LIN {X 0,Y 203.578,Z 1003.73,A -85,B 0,C 180,E1 8716.654,E2 8716.654} C_VEL
LIN {X 0,Y 203.632,Z 1006.005,A -85,B 0,C 180,E1 8711.685,E2 8711.685} C_VEL
LIN {X 0,Y 204.624,Z 1006.572,A -85,B 0,C 180,E1 8706.685,E2 8706.685} C_VEL
LIN {X 0,Y 206.666,Z 1005.305,A -85,B 0,C 180,E1 8701.698,E2 8701.698} C_VEL
LIN {X 0,Y 209.886,Z 1002.177,A -85,B 0,C 180,E1 8696.782,E2 8696.782} C_VEL
LIN {X 0,Y 214.071,Z 997.405,A -85,B 0,C 180,E1 8692.277,E2 8692.277} C_VEL
LIN {X 0,Y 219.005,Z 991.1,A -85,B 0,C 180,E1 8688.199,E2 8688.199} C_VEL
LIN {X 0,Y 224.873,Z 982.735,A -85,B 0,C 180,E1 8684.287,E2 8684.287} C_VEL
LIN {X 0,Y 231.227,Z 972.677,A -85,B 0,C 180,E1 8680.765,E2 8680.765} C_VEL
LIN {X 0,Y 237.626,Z 961.261,A -85,B 0,C 180,E1 8677.717,E2 8677.717} C_VEL
LIN {X 0,Y 243.815,Z 948.504,A -85,B 0,C 180,E1 8675.103,E2 8675.103} C_VEL
LIN {X 0,Y 249.813,Z 934.055,A -85,B 0,C 180,E1 8672.807,E2 8672.807} C_VEL
LIN {X 0,Y 254.885,Z 919.39,A -85,B 0,C 180,E1 8671.005,E2 8671.005} C_VEL
LIN {X 0,Y 259.318,Z 903.23,A -85,B 0,C 180,E1 8669.492,E2 8669.492} C_VEL
LIN {X 0,Y 262.776,Z 886.237,A -85,B 0,C 180,E1 8668.313,E2 8668.313} C_VEL
LIN {X 0,Y 265.149,Z 868.666,A -85,B 0,C 180,E1 8667.459,E2 8667.459} C_VEL
LIN {X 0,Y 267.85,Z 833.08,A -85,B 0,C 180,E1 8666.452,E2 8666.452} C_VEL
LIN {X 0,Y 269.767,Z 808.526,A -85,B 0,C 180,E1 8665.844,E2 8665.844} C_VEL
LIN {X 0,Y 269.834,Z 800.953,A -85,B 0,C 180,E1 8665.478,E2 8665.478} C_VEL
LIN {X 0,Y 268.193,Z 781.182,A -85,B 0,C 180,E1 8663.856,E2 8663.856} C_VEL
LIN {X 0,Y 268.351,Z 774.67,A -85,B 0,C 180,E1 8663.562,E2 8663.562} C_VEL
LIN {X 0,Y 268.8,Z 767.997,A -85,B 0,C 180,E1 8663.367,E2 8663.367} C_VEL
LIN {X 0,Y 263.509,Z 757.018,A -85,B 0,C 180,E1 8660.606,E2 8660.606} C_VEL
LIN {X 0,Y 258.076,Z 747.072,A -85,B 0,C 180,E1 8657.415,E2 8657.415} C_VEL
LIN {X 0,Y 253.684,Z 739.87,A -85,B 0,C 180,E1 8654.378,E2 8654.378} C_VEL
LIN {X 0,Y 250.818,Z 735.384,A -85,B 0,C 180,E1 8652.081,E2 8652.081} C_VEL
LIN {X 0,Y 246.984,Z 729.389,A -85,B 0,C 180,E1 8648.263,E2 8648.263} C_VEL
LIN {X 0,Y 243.777,Z 724.701,A -85,B 0,C 180,E1 8643.763,E2 8643.763} C_VEL
LIN {X 0,Y 241.598,Z 721.587,A -85,B 0,C 180,E1 8637.391,E2 8637.391} C_VEL
LIN {X 0,Y 241.91,Z 721.898,A -85,B 0,C 180,E1 8631.922,E2 8631.922} C_VEL
LIN {X 0,Y 245.181,Z 726.188,A -85,B 0,C 180,E1 8624.992,E2 8624.992} C_VEL
LIN {X 0,Y 249.877,Z 733.151,A -85,B 0,C 180,E1 8619.75,E2 8619.75} C_VEL
LIN {X 0,Y 254.492,Z 740.242,A -85,B 0,C 180,E1 8616.007,E2 8616.007} C_VEL
LIN {X 0,Y 259.061,Z 747.772,A -85,B 0,C 180,E1 8612.97,E2 8612.97} C_VEL
LIN {X 0,Y 263.465,Z 755.393,A -85,B 0,C 180,E1 8610.439,E2 8610.439} C_VEL
LIN {X 0,Y 268.804,Z 765.811,A -85,B 0,C 180,E1 8607.677,E2 8607.677} C_VEL
LIN {X 0,Y 269.518,Z 767.79,A -85,B 0,C 180,E1 8607.302,E2 8607.302} C_VEL
LIN {X 0,Y 259.299,Z 896.401,A -85,B 0,C 180,E1 8604.125,E2 8604.125} C_VEL
LIN {X 0,Y 256.355,Z 915.058,A -85,B 0,C 180,E1 8603.402,E2 8603.402} C_VEL
LIN {X 0,Y 252.244,Z 932.623,A -85,B 0,C 180,E1 8602.444,E2 8602.444} C_VEL
LIN {X 0,Y 246.71,Z 950.675,A -85,B 0,C 180,E1 8601.089,E2 8601.089} C_VEL
LIN {X 0,Y 240.772,Z 966.702,A -85,B 0,C 180,E1 8599.459,E2 8599.459} C_VEL
LIN {X 0,Y 234.223,Z 981.979,A -85,B 0,C 180,E1 8597.423,E2 8597.423} C_VEL
LIN {X 0,Y 227.206,Z 996.499,A -85,B 0,C 180,E1 8594.917,E2 8594.917} C_VEL
LIN {X 0,Y 220.048,Z 1010.012,A -85,B 0,C 180,E1 8591.908,E2 8591.908} C_VEL
LIN {X 0,Y 212.964,Z 1022.543,A -85,B 0,C 180,E1 8588.296,E2 8588.296} C_VEL
LIN {X 0,Y 206.391,Z 1033.8,A -85,B 0,C 180,E1 8584.065,E2 8584.065} C_VEL
LIN {X 0,Y 201.054,Z 1043.16,A -85,B 0,C 180,E1 8579.493,E2 8579.493} C_VEL
LIN {X 0,Y 196.839,Z 1051.262,A -85,B 0,C 180,E1 8574.295,E2 8574.295} C_VEL
LIN {X 0,Y 194.203,Z 1057.772,A -85,B 0,C 180,E1 8568.614,E2 8568.614} C_VEL
LIN {X 0,Y 193.286,Z 1062.33,A -85,B 0,C 180,E1 8562.851,E2 8562.851} C_VEL
LIN {X 0,Y 193.748,Z 1064.894,A -85,B 0,C 180,E1 8557.412,E2 8557.412} C_VEL
LIN {X 0,Y 194.69,Z 1065.679,A -85,B 0,C 180,E1 8552.648,E2 8552.648} C_VEL
LIN {X 0,Y 194.99,Z 1065.259,A -85,B 0,C 180,E1 8549.118,E2 8549.118} C_VEL
LIN {X 0,Y 194.449,Z 1063.524,A -85,B 0,C 180,E1 8544.984,E2 8544.984} C_VEL
LIN {X 0,Y 193.509,Z 1061.492,A -85,B 0,C 180,E1 8539.279,E2 8539.279} C_VEL
LIN {X 0,Y 193.709,Z 1057.837,A -85,B 0,C 180,E1 8534.122,E2 8534.122} C_VEL
LIN {X 0,Y 195.37,Z 1051.854,A -85,B 0,C 180,E1 8528.692,E2 8528.692} C_VEL
LIN {X 0,Y 198.492,Z 1044.215,A -85,B 0,C 180,E1 8523.686,E2 8523.686} C_VEL
LIN {X 0,Y 203.06,Z 1034.434,A -85,B 0,C 180,E1 8518.867,E2 8518.867} C_VEL
LIN {X 0,Y 208.337,Z 1023.844,A -85,B 0,C 180,E1 8514.836,E2 8514.836} C_VEL
LIN {X 0,Y 214.759,Z 1011.017,A -85,B 0,C 180,E1 8511.058,E2 8511.058} C_VEL
LIN {X 0,Y 221.183,Z 997.712,A -85,B 0,C 180,E1 8508.006,E2 8508.006} C_VEL
LIN {X 0,Y 228.022,Z 982.335,A -85,B 0,C 180,E1 8505.264,E2 8505.264} C_VEL
LIN {X 0,Y 234.291,Z 966.649,A -85,B 0,C 180,E1 8503.133,E2 8503.133} C_VEL
LIN {X 0,Y 240.05,Z 949.931,A -85,B 0,C 180,E1 8501.431,E2 8501.431} C_VEL
LIN {X 0,Y 244.754,Z 933.123,A -85,B 0,C 180,E1 8500.21,E2 8500.21} C_VEL
LIN {X 0,Y 248.664,Z 914.35,A -85,B 0,C 180,E1 8499.236,E2 8499.236} C_VEL
LIN {X 0,Y 268.436,Z 803.055,A -85,B 0,C 180,E1 8494.981,E2 8494.981} C_VEL
LIN {X 0,Y 273.515,Z 775.803,A -85,B 0,C 180,E1 8493.883,E2 8493.883} C_VEL
LIN {X 0,Y 274.688,Z 769.516,A -85,B 0,C 180,E1 8493.533,E2 8493.533} C_VEL
LIN {X 0,Y 276.759,Z 763.473,A -85,B 0,C 180,E1 8492.948,E2 8492.948} C_VEL
LIN {X 0,Y 277.255,Z 762.029,A -85,B 0,C 180,E1 8492.448,E2 8492.448} C_VEL
LIN {X 0,Y 276.155,Z 764.633,A -85,B 0,C 180,E1 8490.216,E2 8490.216} C_VEL
LIN {X 0,Y 276.372,Z 769.354,A -85,B 0,C 180,E1 8488.054,E2 8488.054} C_VEL
LIN {X 0,Y 276.354,Z 770.749,A -85,B 0,C 180,E1 8487.719,E2 8487.719} C_VEL
LIN {X 0,Y 276.091,Z 773.303,A -85,B 0,C 180,E1 8487.445,E2 8487.445} C_VEL
LIN {X 0,Y 260.146,Z 869.807,A -85,B 0,C 180,E1 8483.989,E2 8483.989} C_VEL
LIN {X 0,Y 255.611,Z 901.484,A -85,B 0,C 180,E1 8482.427,E2 8482.427} C_VEL
LIN {X 0,Y 252.75,Z 916.861,A -85,B 0,C 180,E1 8481.342,E2 8481.342} C_VEL
LIN {X 0,Y 248.618,Z 932.379,A -85,B 0,C 180,E1 8479.866,E2 8479.866} C_VEL
LIN {X 0,Y 243.925,Z 946.223,A -85,B 0,C 180,E1 8478.151,E2 8478.151} C_VEL
LIN {X 0,Y 238.087,Z 960.158,A -85,B 0,C 180,E1 8475.907,E2 8475.907} C_VEL
LIN {X 0,Y 232.173,Z 971.846,A -85,B 0,C 180,E1 8473.447,E2 8473.447} C_VEL
LIN {X 0,Y 226.238,Z 982.029,A -85,B 0,C 180,E1 8470.697,E2 8470.697} C_VEL
LIN {X 0,Y 219.74,Z 991.542,A -85,B 0,C 180,E1 8467.273,E2 8467.273} C_VEL
LIN {X 0,Y 214.041,Z 998.695,A -85,B 0,C 180,E1 8463.749,E2 8463.749} C_VEL
LIN {X 0,Y 208.667,Z 1004.435,A -85,B 0,C 180,E1 8459.725,E2 8459.725} C_VEL
LIN {X 0,Y 204.19,Z 1008.247,A -85,B 0,C 180,E1 8455.506,E2 8455.506} C_VEL
LIN {X 0,Y 200.448,Z 1010.368,A -85,B 0,C 180,E1 8450.815,E2 8450.815} C_VEL
LIN {X 0,Y 197.801,Z 1010.466,A -85,B 0,C 180,E1 8446.061,E2 8446.061} C_VEL
LIN {X 0,Y 196.221,Z 1008.801,A -85,B 0,C 180,E1 8441.404,E2 8441.404} C_VEL
LIN {X 0,Y 195.451,Z 1005.065,A -85,B 0,C 180,E1 8436.482,E2 8436.482} C_VEL
LIN {X 0,Y 195.491,Z 999.785,A -85,B 0,C 180,E1 8431.93,E2 8431.93} C_VEL
LIN {X 0,Y 196.255,Z 992.329,A -85,B 0,C 180,E1 8427.313,E2 8427.313} C_VEL
LIN {X 0,Y 197.544,Z 983.866,A -85,B 0,C 180,E1 8423.326,E2 8423.326} C_VEL
LIN {X 0,Y 199.467,Z 973.093,A -85,B 0,C 180,E1 8419.333,E2 8419.333} C_VEL
LIN {X 0,Y 201.823,Z 960.491,A -85,B 0,C 180,E1 8415.69,E2 8415.69} C_VEL
LIN {X 0,Y 204.168,Z 947.545,A -85,B 0,C 180,E1 8412.727,E2 8412.727} C_VEL
LIN {X 0,Y 206.602,Z 932.888,A -85,B 0,C 180,E1 8410.066,E2 8410.066} C_VEL
LIN {X 0,Y 208.893,Z 916.417,A -85,B 0,C 180,E1 8407.784,E2 8407.784} C_VEL
LIN {X 0,Y 210.657,Z 900.18,A -85,B 0,C 180,E1 8406.102,E2 8406.102} C_VEL
LIN {X 0,Y 211.969,Z 882.792,A -85,B 0,C 180,E1 8404.823,E2 8404.823} C_VEL
LIN {X 0,Y 214.763,Z 828.021,A -85,B 0,C 180,E1 8402.341,E2 8402.341} C_VEL
LIN {X 0,Y 217.097,Z 797.981,A -85,B 0,C 180,E1 8400.978,E2 8400.978} C_VEL
LIN {X 0,Y 218.251,Z 792.429,A -85,B 0,C 180,E1 8400.462,E2 8400.462} C_VEL
LIN {X 0,Y 220.656,Z 789.756,A -85,B 0,C 180,E1 8399.866,E2 8399.866} C_VEL
LIN {X 0,Y 223.732,Z 783.211,A -85,B 0,C 180,E1 8399.37,E2 8399.37} C_VEL
LIN {X 0,Y 228.317,Z 768.728,A -85,B 0,C 180,E1 8398.869,E2 8398.869} C_VEL
LIN {X 0,Y 232.213,Z 755.083,A -85,B 0,C 180,E1 8398.519,E2 8398.519} C_VEL
LIN {X 0,Y 236.759,Z 749.133,A -85,B 0,C 180,E1 8397.714,E2 8397.714} C_VEL
LIN {X 0,Y 237.715,Z 747.772,A -85,B 0,C 180,E1 8397.554,E2 8397.554} C_VEL
LIN {X 0,Y 238.404,Z 755.137,A -85,B 0,C 180,E1 8397.101,E2 8397.101} C_VEL
LIN {X 0,Y 232.035,Z 861.838,A -85,B 0,C 180,E1 8394.081,E2 8394.081} C_VEL
LIN {X 0,Y 230.476,Z 879.542,A -85,B 0,C 180,E1 8393.202,E2 8393.202} C_VEL
LIN {X 0,Y 228.187,Z 895.686,A -85,B 0,C 180,E1 8392.003,E2 8392.003} C_VEL
LIN {X 0,Y 224.933,Z 912.565,A -85,B 0,C 180,E1 8390.288,E2 8390.288} C_VEL
LIN {X 0,Y 221.154,Z 928.279,A -85,B 0,C 180,E1 8388.178,E2 8388.178} C_VEL
LIN {X 0,Y 217.076,Z 942.488,A -85,B 0,C 180,E1 8385.705,E2 8385.705} C_VEL
LIN {X 0,Y 212.77,Z 955.748,A -85,B 0,C 180,E1 8382.761,E2 8382.761} C_VEL
LIN {X 0,Y 208.516,Z 967.742,A -85,B 0,C 180,E1 8379.384,E2 8379.384} C_VEL
LIN {X 0,Y 204.574,Z 978.262,A -85,B 0,C 180,E1 8375.61,E2 8375.61} C_VEL
LIN {X 0,Y 201.023,Z 987.567,A -85,B 0,C 180,E1 8371.263,E2 8371.263} C_VEL
LIN {X 0,Y 198.271,Z 995.222,A -85,B 0,C 180,E1 8366.531,E2 8366.531} C_VEL
LIN {X 0,Y 196.546,Z 1000.808,A -85,B 0,C 180,E1 8361.812,E2 8361.812} C_VEL
LIN {X 0,Y 195.657,Z 1004.859,A -85,B 0,C 180,E1 8356.706,E2 8356.706} C_VEL
LIN {X 0,Y 195.725,Z 1007.171,A -85,B 0,C 180,E1 8351.536,E2 8351.536} C_VEL
LIN {X 0,Y 196.795,Z 1007.783,A -85,B 0,C 180,E1 8346.337,E2 8346.337} C_VEL
LIN {X 0,Y 198.981,Z 1006.591,A -85,B 0,C 180,E1 8341.159,E2 8341.159} C_VEL
LIN {X 0,Y 202.406,Z 1003.52,A -85,B 0,C 180,E1 8336.069,E2 8336.069} C_VEL
LIN {X 0,Y 206.835,Z 998.812,A -85,B 0,C 180,E1 8331.421,E2 8331.421} C_VEL
LIN {X 0,Y 212.033,Z 992.609,A -85,B 0,C 180,E1 8327.232,E2 8327.232} C_VEL
LIN {X 0,Y 218.188,Z 984.347,A -85,B 0,C 180,E1 8323.229,E2 8323.229} C_VEL
LIN {X 0,Y 224.746,Z 974.521,A -85,B 0,C 180,E1 8319.679,E2 8319.679} C_VEL
LIN {X 0,Y 231.49,Z 963.14,A -85,B 0,C 180,E1 8316.547,E2 8316.547} C_VEL
LIN {X 0,Y 238.009,Z 950.434,A -85,B 0,C 180,E1 8313.872,E2 8313.872} C_VEL
LIN {X 0,Y 244.144,Z 936.403,A -85,B 0,C 180,E1 8311.589,E2 8311.589} C_VEL
LIN {X 0,Y 249.711,Z 921.122,A -85,B 0,C 180,E1 8309.672,E2 8309.672} C_VEL
LIN {X 0,Y 254.364,Z 905.152,A -85,B 0,C 180,E1 8308.145,E2 8308.145} C_VEL
LIN {X 0,Y 258.014,Z 888.279,A -85,B 0,C 180,E1 8306.949,E2 8306.949} C_VEL
LIN {X 0,Y 260.608,Z 870.365,A -85,B 0,C 180,E1 8306.056,E2 8306.056} C_VEL
LIN {X 0,Y 262.922,Z 841.507,A -85,B 0,C 180,E1 8305.196,E2 8305.196} C_VEL
LIN {X 0,Y 268.351,Z 774.67,A -85,B 0,C 180,E1 8303.562,E2 8303.562} C_VEL
LIN {X 0,Y 268.12,Z 771.832,A -85,B 0,C 180,E1 8303.321,E2 8303.321} C_VEL
LIN {X 0,Y 266.748,Z 768.797,A -85,B 0,C 180,E1 8302.625,E2 8302.625} C_VEL
LIN {X 0,Y 263.914,Z 766.213,A -85,B 0,C 180,E1 8301.332,E2 8301.332} C_VEL
LIN {X 0,Y 260.671,Z 763.319,A -85,B 0,C 180,E1 8299.747,E2 8299.747} C_VEL
LIN {X 0,Y 260.14,Z 762.462,A -85,B 0,C 180,E1 8299.45,E2 8299.45} C_VEL
LIN {X 0,Y 255.618,Z 753.768,A -85,B 0,C 180,E1 8296.592,E2 8296.592} C_VEL
LIN {X 0,Y 251.564,Z 746.869,A -85,B 0,C 180,E1 8293.621,E2 8293.621} C_VEL
LIN {X 0,Y 248.889,Z 742.531,A -85,B 0,C 180,E1 8291.353,E2 8291.353} C_VEL
LIN {X 0,Y 245.454,Z 736.952,A -85,B 0,C 180,E1 8287.726,E2 8287.726} C_VEL
LIN {X 0,Y 242.497,Z 732.417,A -85,B 0,C 180,E1 8283.31,E2 8283.31} C_VEL
LIN {X 0,Y 240.565,Z 729.488,A -85,B 0,C 180,E1 8277.142,E2 8277.142} C_VEL
LIN {X 0,Y 240.896,Z 729.875,A -85,B 0,C 180,E1 8271.888,E2 8271.888} C_VEL
LIN {X 0,Y 243.919,Z 734.075,A -85,B 0,C 180,E1 8265.277,E2 8265.277} C_VEL
LIN {X 0,Y 248.264,Z 740.711,A -85,B 0,C 180,E1 8260.227,E2 8260.227} C_VEL
LIN {X 0,Y 252.592,Z 747.658,A -85,B 0,C 180,E1 8256.559,E2 8256.559} C_VEL
LIN {X 0,Y 256.823,Z 754.954,A -85,B 0,C 180,E1 8253.59,E2 8253.59} C_VEL
LIN {X 0,Y 261.285,Z 762.982,A -85,B 0,C 180,E1 8250.923,E2 8250.923} C_VEL
LIN {X 0,Y 265.322,Z 771.367,A -85,B 0,C 180,E1 8248.717,E2 8248.717} C_VEL
LIN {X 0,Y 255.038,Z 895.526,A -85,B 0,C 180,E1 8245.649,E2 8245.649} C_VEL
LIN {X 0,Y 251.997,Z 914.175,A -85,B 0,C 180,E1 8244.931,E2 8244.931} C_VEL
LIN {X 0,Y 247.449,Z 932.835,A -85,B 0,C 180,E1 8243.913,E2 8243.913} C_VEL
LIN {X 0,Y 242.101,Z 949.634,A -85,B 0,C 180,E1 8242.655,E2 8242.655} C_VEL
LIN {X 0,Y 235.949,Z 965.673,A -85,B 0,C 180,E1 8241.04,E2 8241.04} C_VEL
LIN {X 0,Y 229.144,Z 980.95,A -85,B 0,C 180,E1 8239.014,E2 8239.014} C_VEL
LIN {X 0,Y 221.852,Z 995.407,A -85,B 0,C 180,E1 8236.519,E2 8236.519} C_VEL
LIN {X 0,Y 214.049,Z 1009.428,A -85,B 0,C 180,E1 8233.366,E2 8233.366} C_VEL
LIN {X 0,Y 206.548,Z 1021.914,A -85,B 0,C 180,E1 8229.675,E2 8229.675} C_VEL
LIN {X 0,Y 199.783,Z 1032.778,A -85,B 0,C 180,E1 8225.488,E2 8225.488} C_VEL
LIN {X 0,Y 193.93,Z 1042.278,A -85,B 0,C 180,E1 8220.691,E2 8220.691} C_VEL
LIN {X 0,Y 189.366,Z 1050.289,A -85,B 0,C 180,E1 8215.32,E2 8215.32} C_VEL
LIN {X 0,Y 186.435,Z 1056.73,A -85,B 0,C 180,E1 8209.42,E2 8209.42} C_VEL
LIN {X 0,Y 185.341,Z 1061.223,A -85,B 0,C 180,E1 8203.412,E2 8203.412} C_VEL
LIN {X 0,Y 185.749,Z 1063.725,A -85,B 0,C 180,E1 8197.733,E2 8197.733} C_VEL
LIN {X 0,Y 186.751,Z 1064.458,A -85,B 0,C 180,E1 8192.761,E2 8192.761} C_VEL
LIN {X 0,Y 187.081,Z 1064.008,A -85,B 0,C 180,E1 8189.08,E2 8189.08} C_VEL
LIN {X 0,Y 186.484,Z 1062.177,A -85,B 0,C 180,E1 8184.77,E2 8184.77} C_VEL
LIN {X 0,Y 185.543,Z 1060.5,A -85,B 0,C 180,E1 8179.128,E2 8179.128} C_VEL
LIN {X 0,Y 185.831,Z 1056.902,A -85,B 0,C 180,E1 8173.43,E2 8173.43} C_VEL
LIN {X 0,Y 187.608,Z 1051.546,A -85,B 0,C 180,E1 8168.022,E2 8168.022} C_VEL
LIN {X 0,Y 191.174,Z 1043.948,A -85,B 0,C 180,E1 8162.596,E2 8162.596} C_VEL
LIN {X 0,Y 195.809,Z 1035.264,A -85,B 0,C 180,E1 8157.922,E2 8157.922} C_VEL
LIN {X 0,Y 201.824,Z 1024.535,A -85,B 0,C 180,E1 8153.522,E2 8153.522} C_VEL
LIN {X 0,Y 208.687,Z 1012.412,A -85,B 0,C 180,E1 8149.698,E2 8149.698} C_VEL
LIN {X 0,Y 216.326,Z 998.234,A -85,B 0,C 180,E1 8146.291,E2 8146.291} C_VEL
LIN {X 0,Y 223.322,Z 984.22,A -85,B 0,C 180,E1 8143.691,E2 8143.691} C_VEL
LIN {X 0,Y 230.618,Z 967.927,A -85,B 0,C 180,E1 8141.404,E2 8141.404} C_VEL
LIN {X 0,Y 236.718,Z 952.148,A -85,B 0,C 180,E1 8139.758,E2 8139.758} C_VEL
LIN {X 0,Y 242.101,Z 935.373,A -85,B 0,C 180,E1 8138.498,E2 8138.498} C_VEL
LIN {X 0,Y 246.595,Z 916.793,A -85,B 0,C 180,E1 8137.514,E2 8137.514} C_VEL
LIN {X 0,Y 253.262,Z 880.318,A -85,B 0,C 180,E1 8136.065,E2 8136.065} C_VEL
LIN {X 0,Y 270.986,Z 787.896,A -85,B 0,C 180,E1 8132.689,E2 8132.689} C_VEL
LIN {X 0,Y 274.114,Z 772.366,A -85,B 0,C 180,E1 8131.977,E2 8131.977} C_VEL
LIN {X 0,Y 274.515,Z 770.48,A -85,B 0,C 180,E1 8131.791,E2 8131.791} C_VEL
LIN {X 0,Y 274.43,Z 774.056,A -85,B 0,C 180,E1 8129.703,E2 8129.703} C_VEL
LIN {X 0,Y 274.437,Z 775.934,A -85,B 0,C 180,E1 8129.019,E2 8129.019} C_VEL
LIN {X 0,Y 257.896,Z 870.774,A -85,B 0,C 180,E1 8125.674,E2 8125.674} C_VEL
LIN {X 0,Y 252.941,Z 902.761,A -85,B 0,C 180,E1 8124.102,E2 8124.102} C_VEL
LIN {X 0,Y 249.734,Z 918.743,A -85,B 0,C 180,E1 8122.977,E2 8122.977} C_VEL
LIN {X 0,Y 245.337,Z 934.072,A -85,B 0,C 180,E1 8121.517,E2 8121.517} C_VEL
LIN {X 0,Y 240.351,Z 947.81,A -85,B 0,C 180,E1 8119.818,E2 8119.818} C_VEL
LIN {X 0,Y 233.955,Z 962.022,A -85,B 0,C 180,E1 8117.522,E2 8117.522} C_VEL
LIN {X 0,Y 227.02,Z 974.708,A -85,B 0,C 180,E1 8114.8,E2 8114.8} C_VEL
LIN {X 0,Y 220.693,Z 984.536,A -85,B 0,C 180,E1 8112.028,E2 8112.028} C_VEL
LIN {X 0,Y 213.872,Z 993.716,A -85,B 0,C 180,E1 8108.603,E2 8108.603} C_VEL
LIN {X 0,Y 207.285,Z 1001.173,A -85,B 0,C 180,E1 8104.703,E2 8104.703} C_VEL
LIN {X 0,Y 201.577,Z 1006.585,A -85,B 0,C 180,E1 8100.568,E2 8100.568} C_VEL
LIN {X 0,Y 196.529,Z 1010.278,A -85,B 0,C 180,E1 8095.915,E2 8095.915} C_VEL
LIN {X 0,Y 192.812,Z 1011.909,A -85,B 0,C 180,E1 8091.35,E2 8091.35} C_VEL
LIN {X 0,Y 189.944,Z 1011.756,A -85,B 0,C 180,E1 8086.297,E2 8086.297} C_VEL
LIN {X 0,Y 188.266,Z 1009.727,A -85,B 0,C 180,E1 8081.418,E2 8081.418} C_VEL
LIN {X 0,Y 187.491,Z 1005.848,A -85,B 0,C 180,E1 8076.423,E2 8076.423} C_VEL
LIN {X 0,Y 187.545,Z 1000.16,A -85,B 0,C 180,E1 8071.604,E2 8071.604} C_VEL
LIN {X 0,Y 188.331,Z 992.822,A -85,B 0,C 180,E1 8067.018,E2 8067.018} C_VEL
LIN {X 0,Y 189.761,Z 983.773,A -85,B 0,C 180,E1 8062.703,E2 8062.703} C_VEL
LIN {X 0,Y 191.624,Z 973.621,A -85,B 0,C 180,E1 8058.894,E2 8058.894} C_VEL
LIN {X 0,Y 194.087,Z 960.838,A -85,B 0,C 180,E1 8055.107,E2 8055.107} C_VEL
LIN {X 0,Y 196.671,Z 946.905,A -85,B 0,C 180,E1 8051.884,E2 8051.884} C_VEL
LIN {X 0,Y 199.111,Z 932.453,A -85,B 0,C 180,E1 8049.252,E2 8049.252} C_VEL
LIN {X 0,Y 201.448,Z 916.135,A -85,B 0,C 180,E1 8046.955,E2 8046.955} C_VEL
LIN {X 0,Y 203.406,Z 898.223,A -85,B 0,C 180,E1 8045.109,E2 8045.109} C_VEL
LIN {X 0,Y 204.686,Z 880.46,A -85,B 0,C 180,E1 8043.857,E2 8043.857} C_VEL
LIN {X 0,Y 206.821,Z 840.303,A -85,B 0,C 180,E1 8041.878,E2 8041.878} C_VEL
LIN {X 0,Y 207.906,Z 834.54,A -85,B 0,C 180,E1 8041.317,E2 8041.317} C_VEL
LIN {X 0,Y 210.557,Z 831.512,A -85,B 0,C 180,E1 8040.604,E2 8040.604} C_VEL
LIN {X 0,Y 213.729,Z 824.641,A -85,B 0,C 180,E1 8040.064,E2 8040.064} C_VEL
LIN {X 0,Y 218.392,Z 809.936,A -85,B 0,C 180,E1 8039.521,E2 8039.521} C_VEL
LIN {X 0,Y 221.875,Z 797.999,A -85,B 0,C 180,E1 8039.176,E2 8039.176} C_VEL
LIN {X 0,Y 225.197,Z 793.883,A -85,B 0,C 180,E1 8038.531,E2 8038.531} C_VEL
LIN {X 0,Y 228.812,Z 786.166,A -85,B 0,C 180,E1 8037.996,E2 8037.996} C_VEL
LIN {X 0,Y 230.951,Z 780.277,A -85,B 0,C 180,E1 8037.746,E2 8037.746} C_VEL
LIN {X 0,Y 225.842,Z 863.105,A -85,B 0,C 180,E1 8035.328,E2 8035.328} C_VEL
LIN {X 0,Y 224.174,Z 880.79,A -85,B 0,C 180,E1 8034.42,E2 8034.42} C_VEL
LIN {X 0,Y 221.612,Z 897.765,A -85,B 0,C 180,E1 8033.112,E2 8033.112} C_VEL
LIN {X 0,Y 218.227,Z 914.383,A -85,B 0,C 180,E1 8031.362,E2 8031.362} C_VEL
LIN {X 0,Y 214.285,Z 929.924,A -85,B 0,C 180,E1 8029.202,E2 8029.202} C_VEL
LIN {X 0,Y 209.94,Z 944.287,A -85,B 0,C 180,E1 8026.605,E2 8026.605} C_VEL
LIN {X 0,Y 205.377,Z 957.66,A -85,B 0,C 180,E1 8023.515,E2 8023.515} C_VEL
LIN {X 0,Y 200.964,Z 969.515,A -85,B 0,C 180,E1 8020.029,E2 8020.029} C_VEL
LIN {X 0,Y 196.868,Z 979.869,A -85,B 0,C 180,E1 8016.123,E2 8016.123} C_VEL
LIN {X 0,Y 193.309,Z 988.784,A -85,B 0,C 180,E1 8011.779,E2 8011.779} C_VEL
LIN {X 0,Y 190.493,Z 996.248,A -85,B 0,C 180,E1 8006.992,E2 8006.992} C_VEL
LIN {X 0,Y 188.669,Z 1001.879,A -85,B 0,C 180,E1 8002.081,E2 8002.081} C_VEL
LIN {X 0,Y 187.736,Z 1005.979,A -85,B 0,C 180,E1 7996.762,E2 7996.762} C_VEL
LIN {X 0,Y 187.821,Z 1008.336,A -85,B 0,C 180,E1 7991.368,E2 7991.368} C_VEL
LIN {X 0,Y 188.973,Z 1008.994,A -85,B 0,C 180,E1 7985.959,E2 7985.959} C_VEL
LIN {X 0,Y 191.316,Z 1007.877,A -85,B 0,C 180,E1 7980.577,E2 7980.577} C_VEL
LIN {X 0,Y 194.961,Z 1004.863,A -85,B 0,C 180,E1 7975.302,E2 7975.302} C_VEL
LIN {X 0,Y 199.716,Z 1000.15,A -85,B 0,C 180,E1 7970.444,E2 7970.444} C_VEL
LIN {X 0,Y 205.524,Z 993.628,A -85,B 0,C 180,E1 7965.919,E2 7965.919} C_VEL
LIN {X 0,Y 212.043,Z 985.323,A -85,B 0,C 180,E1 7961.84,E2 7961.84} C_VEL
LIN {X 0,Y 218.952,Z 975.464,A -85,B 0,C 180,E1 7958.239,E2 7958.239} C_VEL
LIN {X 0,Y 226.021,Z 964.051,A -85,B 0,C 180,E1 7955.077,E2 7955.077} C_VEL
LIN {X 0,Y 232.713,Z 951.563,A -85,B 0,C 180,E1 7952.43,E2 7952.43} C_VEL
LIN {X 0,Y 238.91,Z 938.055,A -85,B 0,C 180,E1 7950.207,E2 7950.207} C_VEL
LIN {X 0,Y 244.645,Z 923.093,A -85,B 0,C 180,E1 7948.301,E2 7948.301} C_VEL
LIN {X 0,Y 249.3,Z 908.081,A -85,B 0,C 180,E1 7946.828,E2 7946.828} C_VEL
LIN {X 0,Y 253.125,Z 892.027,A -85,B 0,C 180,E1 7945.632,E2 7945.632} C_VEL
LIN {X 0,Y 255.929,Z 874.811,A -85,B 0,C 180,E1 7944.716,E2 7944.716} C_VEL
LIN {X 0,Y 257.849,Z 853.864,A -85,B 0,C 180,E1 7944.004,E2 7944.004} C_VEL
LIN {X 0,Y 264.601,Z 771.729,A -85,B 0,C 180,E1 7941.94,E2 7941.94} C_VEL
LIN {X 0,Y 260.14,Z 762.462,A -85,B 0,C 180,E1 7939.45,E2 7939.45} C_VEL
LIN {X 0,Y 257.969,Z 759.528,A -85,B 0,C 180,E1 7938.219,E2 7938.219} C_VEL
LIN {X 0,Y 254.049,Z 756.875,A -85,B 0,C 180,E1 7935.95,E2 7935.95} C_VEL
LIN {X 0,Y 249.798,Z 754.067,A -85,B 0,C 180,E1 7933.086,E2 7933.086} C_VEL
LIN {X 0,Y 248.674,Z 752.455,A -85,B 0,C 180,E1 7932.153,E2 7932.153} C_VEL
LIN {X 0,Y 245.174,Z 746.515,A -85,B 0,C 180,E1 7928.679,E2 7928.679} C_VEL
LIN {X 0,Y 243.412,Z 743.839,A -85,B 0,C 180,E1 7926.487,E2 7926.487} C_VEL
LIN {X 0,Y 241.283,Z 740.193,A -85,B 0,C 180,E1 7922.95,E2 7922.95} C_VEL
LIN {X 0,Y 239.559,Z 737.429,A -85,B 0,C 180,E1 7917.13,E2 7917.13} C_VEL
LIN {X 0,Y 239.831,Z 737.761,A -85,B 0,C 180,E1 7912.093,E2 7912.093} C_VEL
LIN {X 0,Y 242.611,Z 741.797,A -85,B 0,C 180,E1 7905.684,E2 7905.684} C_VEL
LIN {X 0,Y 246.669,Z 748.274,A -85,B 0,C 180,E1 7900.71,E2 7900.71} C_VEL
LIN {X 0,Y 250.766,Z 755.159,A -85,B 0,C 180,E1 7897.078,E2 7897.078} C_VEL
LIN {X 0,Y 255.195,Z 763.112,A -85,B 0,C 180,E1 7893.847,E2 7893.847} C_VEL
LIN {X 0,Y 260.094,Z 772.731,A -85,B 0,C 180,E1 7890.84,E2 7890.84} C_VEL
LIN {X 0,Y 261.237,Z 775.586,A -85,B 0,C 180,E1 7890.162,E2 7890.162} C_VEL
LIN {X 0,Y 251.007,Z 894.719,A -85,B 0,C 180,E1 7887.23,E2 7887.23} C_VEL
LIN {X 0,Y 247.878,Z 913.35,A -85,B 0,C 180,E1 7886.52,E2 7886.52} C_VEL
LIN {X 0,Y 243.573,Z 930.688,A -85,B 0,C 180,E1 7885.597,E2 7885.597} C_VEL
LIN {X 0,Y 237.687,Z 948.708,A -85,B 0,C 180,E1 7884.279,E2 7884.279} C_VEL
LIN {X 0,Y 230.995,Z 965.461,A -85,B 0,C 180,E1 7882.598,E2 7882.598} C_VEL
LIN {X 0,Y 223.626,Z 981.222,A -85,B 0,C 180,E1 7880.482,E2 7880.482} C_VEL
LIN {X 0,Y 215.74,Z 996.018,A -85,B 0,C 180,E1 7877.861,E2 7877.861} C_VEL
LIN {X 0,Y 207.643,Z 1009.682,A -85,B 0,C 180,E1 7874.67,E2 7874.67} C_VEL
LIN {X 0,Y 199.883,Z 1021.85,A -85,B 0,C 180,E1 7870.941,E2 7870.941} C_VEL
LIN {X 0,Y 192.744,Z 1032.588,A -85,B 0,C 180,E1 7866.623,E2 7866.623} C_VEL
LIN {X 0,Y 186.575,Z 1041.897,A -85,B 0,C 180,E1 7861.68,E2 7861.68} C_VEL
LIN {X 0,Y 181.734,Z 1049.729,A -85,B 0,C 180,E1 7856.112,E2 7856.112} C_VEL
LIN {X 0,Y 178.706,Z 1055.692,A -85,B 0,C 180,E1 7850.296,E2 7850.296} C_VEL
LIN {X 0,Y 177.408,Z 1060.117,A -85,B 0,C 180,E1 7844.024,E2 7844.024} C_VEL
LIN {X 0,Y 177.749,Z 1062.559,A -85,B 0,C 180,E1 7838.083,E2 7838.083} C_VEL
LIN {X 0,Y 178.804,Z 1063.233,A -85,B 0,C 180,E1 7832.884,E2 7832.884} C_VEL
LIN {X 0,Y 179.19,Z 1062.817,A -85,B 0,C 180,E1 7829.36,E2 7829.36} C_VEL
LIN {X 0,Y 178.618,Z 1061.123,A -85,B 0,C 180,E1 7825.13,E2 7825.13} C_VEL
LIN {X 0,Y 178.116,Z 1060.38,A -85,B 0,C 180,E1 7822.581,E2 7822.581} C_VEL
LIN {X 0,Y 177.512,Z 1058.574,A -85,B 0,C 180,E1 7816.978,E2 7816.978} C_VEL
LIN {X 0,Y 178.297,Z 1054.97,A -85,B 0,C 180,E1 7811.358,E2 7811.358} C_VEL
LIN {X 0,Y 180.681,Z 1049.547,A -85,B 0,C 180,E1 7805.825,E2 7805.825} C_VEL
LIN {X 0,Y 185.05,Z 1041.806,A -85,B 0,C 180,E1 7800.191,E2 7800.191} C_VEL
LIN {X 0,Y 190.449,Z 1033.08,A -85,B 0,C 180,E1 7795.458,E2 7795.458} C_VEL
LIN {X 0,Y 197.262,Z 1022.384,A -85,B 0,C 180,E1 7791.058,E2 7791.058} C_VEL
LIN {X 0,Y 204.868,Z 1010.323,A -85,B 0,C 180,E1 7787.281,E2 7787.281} C_VEL
LIN {X 0,Y 213.166,Z 996.322,A -85,B 0,C 180,E1 7783.963,E2 7783.963} C_VEL
LIN {X 0,Y 220.762,Z 982.419,A -85,B 0,C 180,E1 7781.446,E2 7781.446} C_VEL
LIN {X 0,Y 228.579,Z 966.327,A -85,B 0,C 180,E1 7779.263,E2 7779.263} C_VEL
LIN {X 0,Y 235.468,Z 949.795,A -85,B 0,C 180,E1 7777.633,E2 7777.633} C_VEL
LIN {X 0,Y 241.207,Z 932.97,A -85,B 0,C 180,E1 7776.468,E2 7776.468} C_VEL
LIN {X 0,Y 245.944,Z 914.407,A -85,B 0,C 180,E1 7775.538,E2 7775.538} C_VEL
LIN {X 0,Y 270.842,Z 789.655,A -85,B 0,C 180,E1 7771.038,E2 7771.038} C_VEL
LIN {X 0,Y 272.74,Z 780.652,A -85,B 0,C 180,E1 7770.635,E2 7770.635} C_VEL
LIN {X 0,Y 272.63,Z 781.409,A -85,B 0,C 180,E1 7770.526,E2 7770.526} C_VEL
LIN {X 0,Y 256.033,Z 872.09,A -85,B 0,C 180,E1 7767.384,E2 7767.384} C_VEL
LIN {X 0,Y 250.676,Z 904.206,A -85,B 0,C 180,E1 7765.817,E2 7765.817} C_VEL
LIN {X 0,Y 247.339,Z 919.801,A -85,B 0,C 180,E1 7764.733,E2 7764.733} C_VEL
LIN {X 0,Y 242.677,Z 935.145,A -85,B 0,C 180,E1 7763.299,E2 7763.299} C_VEL
LIN {X 0,Y 237.393,Z 948.916,A -85,B 0,C 180,E1 7761.625,E2 7761.625} C_VEL
LIN {X 0,Y 230.614,Z 963.079,A -85,B 0,C 180,E1 7759.37,E2 7759.37} C_VEL
LIN {X 0,Y 223.491,Z 975.333,A -85,B 0,C 180,E1 7756.782,E2 7756.782} C_VEL
LIN {X 0,Y 216.963,Z 984.98,A -85,B 0,C 180,E1 7754.137,E2 7754.137} C_VEL
LIN {X 0,Y 209.554,Z 994.309,A -85,B 0,C 180,E1 7750.724,E2 7750.724} C_VEL
LIN {X 0,Y 202.823,Z 1001.55,A -85,B 0,C 180,E1 7747.079,E2 7747.079} C_VEL
LIN {X 0,Y 196.059,Z 1007.581,A -85,B 0,C 180,E1 7742.63,E2 7742.63} C_VEL
LIN {X 0,Y 190.711,Z 1011.253,A -85,B 0,C 180,E1 7738.197,E2 7738.197} C_VEL
LIN {X 0,Y 186.153,Z 1013.278,A -85,B 0,C 180,E1 7733.213,E2 7733.213} C_VEL
LIN {X 0,Y 182.78,Z 1013.286,A -85,B 0,C 180,E1 7728.002,E2 7728.002} C_VEL
LIN {X 0,Y 180.723,Z 1011.519,A -85,B 0,C 180,E1 7722.948,E2 7722.948} C_VEL
LIN {X 0,Y 179.653,Z 1007.84,A -85,B 0,C 180,E1 7717.761,E2 7717.761} C_VEL
LIN {X 0,Y 179.49,Z 1002.59,A -85,B 0,C 180,E1 7712.819,E2 7712.819} C_VEL
LIN {X 0,Y 180.147,Z 995.165,A -85,B 0,C 180,E1 7707.803,E2 7707.803} C_VEL
LIN {X 0,Y 181.419,Z 986.794,A -85,B 0,C 180,E1 7703.471,E2 7703.471} C_VEL
LIN {X 0,Y 183.39,Z 976.121,A -85,B 0,C 180,E1 7699.136,E2 7699.136} C_VEL
LIN {X 0,Y 185.801,Z 963.933,A -85,B 0,C 180,E1 7695.264,E2 7695.264} C_VEL
LIN {X 0,Y 188.345,Z 950.925,A -85,B 0,C 180,E1 7691.983,E2 7691.983} C_VEL
LIN {X 0,Y 191.016,Z 935.975,A -85,B 0,C 180,E1 7689.038,E2 7689.038} C_VEL
LIN {X 0,Y 193.343,Z 920.771,A -85,B 0,C 180,E1 7686.719,E2 7686.719} C_VEL
LIN {X 0,Y 195.346,Z 904.619,A -85,B 0,C 180,E1 7684.842,E2 7684.842} C_VEL
LIN {X 0,Y 197.013,Z 885.421,A -85,B 0,C 180,E1 7683.275,E2 7683.275} C_VEL
LIN {X 0,Y 197.886,Z 873.416,A -85,B 0,C 180,E1 7682.455,E2 7682.455} C_VEL
LIN {X 0,Y 198.691,Z 870.889,A -85,B 0,C 180,E1 7682.011,E2 7682.011} C_VEL
LIN {X 0,Y 200.957,Z 869.284,A -85,B 0,C 180,E1 7681.358,E2 7681.358} C_VEL
LIN {X 0,Y 203.308,Z 865.478,A -85,B 0,C 180,E1 7680.92,E2 7680.92} C_VEL
LIN {X 0,Y 206.86,Z 855.827,A -85,B 0,C 180,E1 7680.437,E2 7680.437} C_VEL
LIN {X 0,Y 211.443,Z 840.037,A -85,B 0,C 180,E1 7679.94,E2 7679.94} C_VEL
LIN {X 0,Y 214.724,Z 836.133,A -85,B 0,C 180,E1 7679.247,E2 7679.247} C_VEL
LIN {X 0,Y 218.302,Z 828.731,A -85,B 0,C 180,E1 7678.67,E2 7678.67} C_VEL
LIN {X 0,Y 222.824,Z 815.466,A -85,B 0,C 180,E1 7678.149,E2 7678.149} C_VEL
LIN {X 0,Y 219.609,Z 866.491,A -85,B 0,C 180,E1 7676.555,E2 7676.555} C_VEL
LIN {X 0,Y 217.655,Z 884.34,A -85,B 0,C 180,E1 7675.547,E2 7675.547} C_VEL
LIN {X 0,Y 214.892,Z 901.104,A -85,B 0,C 180,E1 7674.171,E2 7674.171} C_VEL
LIN {X 0,Y 211.374,Z 917.183,A -85,B 0,C 180,E1 7672.383,E2 7672.383} C_VEL
LIN {X 0,Y 207.271,Z 932.224,A -85,B 0,C 180,E1 7670.177,E2 7670.177} C_VEL
LIN {X 0,Y 202.557,Z 946.983,A -85,B 0,C 180,E1 7667.377,E2 7667.377} C_VEL
LIN {X 0,Y 197.841,Z 960.084,A -85,B 0,C 180,E1 7664.189,E2 7664.189} C_VEL
LIN {X 0,Y 193.258,Z 971.674,A -85,B 0,C 180,E1 7660.575,E2 7660.575} C_VEL
LIN {X 0,Y 188.903,Z 982.121,A -85,B 0,C 180,E1 7656.383,E2 7656.383} C_VEL
LIN {X 0,Y 185.279,Z 990.829,A -85,B 0,C 180,E1 7651.856,E2 7651.856} C_VEL
LIN {X 0,Y 182.434,Z 998.11,A -85,B 0,C 180,E1 7646.859,E2 7646.859} C_VEL
LIN {X 0,Y 180.54,Z 1003.784,A -85,B 0,C 180,E1 7641.401,E2 7641.401} C_VEL
LIN {X 0,Y 179.75,Z 1007.639,A -85,B 0,C 180,E1 7635.834,E2 7635.834} C_VEL
LIN {X 0,Y 180.053,Z 1009.776,A -85,B 0,C 180,E1 7630.201,E2 7630.201} C_VEL
LIN {X 0,Y 181.51,Z 1010.154,A -85,B 0,C 180,E1 7624.554,E2 7624.554} C_VEL
LIN {X 0,Y 184.249,Z 1008.747,A -85,B 0,C 180,E1 7618.968,E2 7618.968} C_VEL
LIN {X 0,Y 188.391,Z 1005.501,A -85,B 0,C 180,E1 7613.529,E2 7613.529} C_VEL
LIN {X 0,Y 193.588,Z 1000.595,A -85,B 0,C 180,E1 7608.617,E2 7608.617} C_VEL
LIN {X 0,Y 199.804,Z 993.843,A -85,B 0,C 180,E1 7604.075,E2 7604.075} C_VEL
LIN {X 0,Y 207.026,Z 985.033,A -85,B 0,C 180,E1 7599.834,E2 7599.834} C_VEL
LIN {X 0,Y 214.412,Z 974.871,A -85,B 0,C 180,E1 7596.222,E2 7596.222} C_VEL
LIN {X 0,Y 221.602,Z 963.492,A -85,B 0,C 180,E1 7593.18,E2 7593.18} C_VEL
LIN {X 0,Y 228.677,Z 950.588,A -85,B 0,C 180,E1 7590.532,E2 7590.532} C_VEL
LIN {X 0,Y 235.139,Z 936.735,A -85,B 0,C 180,E1 7588.334,E2 7588.334} C_VEL
LIN {X 0,Y 240.836,Z 922.059,A -85,B 0,C 180,E1 7586.535,E2 7586.535} C_VEL
LIN {X 0,Y 245.8,Z 905.891,A -85,B 0,C 180,E1 7585.028,E2 7585.028} C_VEL
LIN {X 0,Y 249.689,Z 888.901,A -85,B 0,C 180,E1 7583.851,E2 7583.851} C_VEL
LIN {X 0,Y 252.39,Z 871.261,A -85,B 0,C 180,E1 7582.992,E2 7582.992} C_VEL
LIN {X 0,Y 255.347,Z 836.957,A -85,B 0,C 180,E1 7582.008,E2 7582.008} C_VEL
LIN {X 0,Y 260.604,Z 775.711,A -85,B 0,C 180,E1 7580.496,E2 7580.496} C_VEL
LIN {X 0,Y 255.752,Z 765.425,A -85,B 0,C 180,E1 7577.52,E2 7577.52} C_VEL
LIN {X 0,Y 252.168,Z 758.682,A -85,B 0,C 180,E1 7574.995,E2 7574.995} C_VEL
LIN {X 0,Y 249.09,Z 753.202,A -85,B 0,C 180,E1 7572.519,E2 7572.519} C_VEL
LIN {X 0,Y 248.674,Z 752.455,A -85,B 0,C 180,E1 7572.153,E2 7572.153} C_VEL
LIN {X 0,Y 247.04,Z 750.586,A -85,B 0,C 180,E1 7570.729,E2 7570.729} C_VEL
LIN {X 0,Y 244.492,Z 750.153,A -85,B 0,C 180,E1 7568.457,E2 7568.457} C_VEL
LIN {X 0,Y 241.618,Z 750.277,A -85,B 0,C 180,E1 7565.314,E2 7565.314} C_VEL
LIN {X 0,Y 240.79,Z 749.314,A -85,B 0,C 180,E1 7564.007,E2 7564.007} C_VEL
LIN {X 0,Y 239.983,Z 747.858,A -85,B 0,C 180,E1 7562.388,E2 7562.388} C_VEL
LIN {X 0,Y 238.529,Z 745.337,A -85,B 0,C 180,E1 7556.877,E2 7556.877} C_VEL
LIN {X 0,Y 238.816,Z 745.745,A -85,B 0,C 180,E1 7552.059,E2 7552.059} C_VEL
LIN {X 0,Y 241.381,Z 749.677,A -85,B 0,C 180,E1 7545.977,E2 7545.977} C_VEL
LIN {X 0,Y 245.09,Z 755.838,A -85,B 0,C 180,E1 7541.199,E2 7541.199} C_VEL
LIN {X 0,Y 248.93,Z 762.597,A -85,B 0,C 180,E1 7537.631,E2 7537.631} C_VEL
LIN {X 0,Y 253.105,Z 770.457,A -85,B 0,C 180,E1 7534.433,E2 7534.433} C_VEL
LIN {X 0,Y 257.37,Z 779.276,A -85,B 0,C 180,E1 7531.663,E2 7531.663} C_VEL
LIN {X 0,Y 247.177,Z 893.893,A -85,B 0,C 180,E1 7528.861,E2 7528.861} C_VEL
LIN {X 0,Y 243.956,Z 912.525,A -85,B 0,C 180,E1 7528.161,E2 7528.161} C_VEL
LIN {X 0,Y 239.151,Z 931.124,A -85,B 0,C 180,E1 7527.177,E2 7527.177} C_VEL
LIN {X 0,Y 233.474,Z 947.846,A -85,B 0,C 180,E1 7525.961,E2 7525.961} C_VEL
LIN {X 0,Y 226.895,Z 963.81,A -85,B 0,C 180,E1 7524.393,E2 7524.393} C_VEL
LIN {X 0,Y 219.455,Z 979.231,A -85,B 0,C 180,E1 7522.374,E2 7522.374} C_VEL
LIN {X 0,Y 211.465,Z 993.715,A -85,B 0,C 180,E1 7519.873,E2 7519.873} C_VEL
LIN {X 0,Y 203.09,Z 1007.323,A -85,B 0,C 180,E1 7516.771,E2 7516.771} C_VEL
LIN {X 0,Y 194.806,Z 1019.681,A -85,B 0,C 180,E1 7513.049,E2 7513.049} C_VEL
LIN {X 0,Y 187.092,Z 1030.582,A -85,B 0,C 180,E1 7508.701,E2 7508.701} C_VEL
LIN {X 0,Y 180.315,Z 1040.032,A -85,B 0,C 180,E1 7503.676,E2 7503.676} C_VEL
LIN {X 0,Y 174.866,Z 1047.992,A -85,B 0,C 180,E1 7497.96,E2 7497.96} C_VEL
LIN {X 0,Y 171.249,Z 1054.17,A -85,B 0,C 180,E1 7491.823,E2 7491.823} C_VEL
LIN {X 0,Y 169.562,Z 1058.612,A -85,B 0,C 180,E1 7485.387,E2 7485.387} C_VEL
LIN {X 0,Y 169.704,Z 1061.285,A -85,B 0,C 180,E1 7478.811,E2 7478.811} C_VEL
LIN {X 0,Y 170.786,Z 1062.002,A -85,B 0,C 180,E1 7473.355,E2 7473.355} C_VEL
LIN {X 0,Y 171.297,Z 1061.624,A -85,B 0,C 180,E1 7469.665,E2 7469.665} C_VEL
LIN {X 0,Y 170.776,Z 1060.144,A -85,B 0,C 180,E1 7465.634,E2 7465.634} C_VEL
LIN {X 0,Y 170.278,Z 1059.054,A -85,B 0,C 180,E1 7462.905,E2 7462.905} C_VEL
LIN {X 0,Y 169.56,Z 1057.715,A -85,B 0,C 180,E1 7457.05,E2 7457.05} C_VEL
LIN {X 0,Y 170.329,Z 1054.566,A -85,B 0,C 180,E1 7451.163,E2 7451.163} C_VEL
LIN {X 0,Y 173.212,Z 1048.985,A -85,B 0,C 180,E1 7444.711,E2 7444.711} C_VEL
LIN {X 0,Y 177.677,Z 1042.13,A -85,B 0,C 180,E1 7439.196,E2 7439.196} C_VEL
LIN {X 0,Y 184.24,Z 1032.805,A -85,B 0,C 180,E1 7433.733,E2 7433.733} C_VEL
LIN {X 0,Y 191.62,Z 1022.578,A -85,B 0,C 180,E1 7429.288,E2 7429.288} C_VEL
LIN {X 0,Y 200.328,Z 1010.173,A -85,B 0,C 180,E1 7425.27,E2 7425.27} C_VEL
LIN {X 0,Y 209.237,Z 996.627,A -85,B 0,C 180,E1 7421.99,E2 7421.99} C_VEL
LIN {X 0,Y 218.277,Z 981.557,A -85,B 0,C 180,E1 7419.272,E2 7419.272} C_VEL
LIN {X 0,Y 226.208,Z 966.613,A -85,B 0,C 180,E1 7417.285,E2 7417.285} C_VEL
LIN {X 0,Y 233.859,Z 949.878,A -85,B 0,C 180,E1 7415.674,E2 7415.674} C_VEL
LIN {X 0,Y 239.873,Z 933.659,A -85,B 0,C 180,E1 7414.589,E2 7414.589} C_VEL
LIN {X 0,Y 245.094,Z 915.41,A -85,B 0,C 180,E1 7413.695,E2 7413.695} C_VEL
LIN {X 0,Y 262.656,Z 831.037,A -85,B 0,C 180,E1 7410.646,E2 7410.646} C_VEL
LIN {X 0,Y 253.368,Z 880.304,A -85,B 0,C 180,E1 7408.835,E2 7408.835} C_VEL
LIN {X 0,Y 248.237,Z 908.823,A -85,B 0,C 180,E1 7407.382,E2 7407.382} C_VEL
LIN {X 0,Y 244.653,Z 923.497,A -85,B 0,C 180,E1 7406.322,E2 7406.322} C_VEL
LIN {X 0,Y 239.397,Z 939.193,A -85,B 0,C 180,E1 7404.818,E2 7404.818} C_VEL
LIN {X 0,Y 233.443,Z 953.039,A -85,B 0,C 180,E1 7403.073,E2 7403.073} C_VEL
LIN {X 0,Y 226.61,Z 966.068,A -85,B 0,C 180,E1 7400.94,E2 7400.94} C_VEL
LIN {X 0,Y 218.448,Z 978.946,A -85,B 0,C 180,E1 7398.134,E2 7398.134} C_VEL
LIN {X 0,Y 210.685,Z 989.16,A -85,B 0,C 180,E1 7395.13,E2 7395.13} C_VEL
LIN {X 0,Y 203.299,Z 997.488,A -85,B 0,C 180,E1 7391.838,E2 7391.838} C_VEL
LIN {X 0,Y 195.843,Z 1004.584,A -85,B 0,C 180,E1 7387.919,E2 7387.919} C_VEL
LIN {X 0,Y 189.157,Z 1009.803,A -85,B 0,C 180,E1 7383.636,E2 7383.636} C_VEL
LIN {X 0,Y 183.028,Z 1013.408,A -85,B 0,C 180,E1 7378.644,E2 7378.644} C_VEL
LIN {X 0,Y 178.346,Z 1014.878,A -85,B 0,C 180,E1 7373.561,E2 7373.561} C_VEL
LIN {X 0,Y 175.019,Z 1014.59,A -85,B 0,C 180,E1 7368.465,E2 7368.465} C_VEL
LIN {X 0,Y 172.815,Z 1012.493,A -85,B 0,C 180,E1 7363.184,E2 7363.184} C_VEL
LIN {X 0,Y 171.688,Z 1008.583,A -85,B 0,C 180,E1 7357.756,E2 7357.756} C_VEL
LIN {X 0,Y 171.523,Z 1002.989,A -85,B 0,C 180,E1 7352.579,E2 7352.579} C_VEL
LIN {X 0,Y 172.167,Z 995.928,A -85,B 0,C 180,E1 7347.703,E2 7347.703} C_VEL
LIN {X 0,Y 173.486,Z 987.384,A -85,B 0,C 180,E1 7343.173,E2 7343.173} C_VEL
LIN {X 0,Y 175.48,Z 976.87,A -85,B 0,C 180,E1 7338.776,E2 7338.776} C_VEL
LIN {X 0,Y 177.979,Z 964.553,A -85,B 0,C 180,E1 7334.746,E2 7334.746} C_VEL
LIN {X 0,Y 180.63,Z 951.37,A -85,B 0,C 180,E1 7331.333,E2 7331.333} C_VEL
LIN {X 0,Y 183.416,Z 936.344,A -85,B 0,C 180,E1 7328.279,E2 7328.279} C_VEL
LIN {X 0,Y 185.999,Z 919.944,A -85,B 0,C 180,E1 7325.735,E2 7325.735} C_VEL
LIN {X 0,Y 187.961,Z 904.427,A -85,B 0,C 180,E1 7323.916,E2 7323.916} C_VEL
LIN {X 0,Y 189.083,Z 894.897,A -85,B 0,C 180,E1 7322.931,E2 7322.931} C_VEL
LIN {X 0,Y 190.044,Z 892.904,A -85,B 0,C 180,E1 7322.378,E2 7322.378} C_VEL
LIN {X 0,Y 192.593,Z 891.712,A -85,B 0,C 180,E1 7321.633,E2 7321.633} C_VEL
LIN {X 0,Y 195.949,Z 887.819,A -85,B 0,C 180,E1 7321.061,E2 7321.061} C_VEL
LIN {X 0,Y 199.843,Z 880.33,A -85,B 0,C 180,E1 7320.715,E2 7320.715} C_VEL
LIN {X 0,Y 201.252,Z 877.243,A -85,B 0,C 180,E1 7320.599,E2 7320.599} C_VEL
LIN {X 0,Y 204.752,Z 874.074,A -85,B 0,C 180,E1 7319.863,E2 7319.863} C_VEL
LIN {X 0,Y 207.971,Z 868.815,A -85,B 0,C 180,E1 7319.364,E2 7319.364} C_VEL
LIN {X 0,Y 211.954,Z 858.49,A -85,B 0,C 180,E1 7318.911,E2 7318.911} C_VEL
LIN {X 0,Y 214.844,Z 848.655,A -85,B 0,C 180,E1 7318.625,E2 7318.625} C_VEL
LIN {X 0,Y 213.252,Z 871.768,A -85,B 0,C 180,E1 7317.744,E2 7317.744} C_VEL
LIN {X 0,Y 211.083,Z 888.934,A -85,B 0,C 180,E1 7316.668,E2 7316.668} C_VEL
LIN {X 0,Y 208.001,Z 905.494,A -85,B 0,C 180,E1 7315.178,E2 7315.178} C_VEL
LIN {X 0,Y 204.1,Z 921.601,A -85,B 0,C 180,E1 7313.227,E2 7313.227} C_VEL
LIN {X 0,Y 199.632,Z 936.743,A -85,B 0,C 180,E1 7310.831,E2 7310.831} C_VEL
LIN {X 0,Y 194.788,Z 950.847,A -85,B 0,C 180,E1 7307.939,E2 7307.939} C_VEL
LIN {X 0,Y 189.936,Z 963.366,A -85,B 0,C 180,E1 7304.637,E2 7304.637} C_VEL
LIN {X 0,Y 184.917,Z 975.312,A -85,B 0,C 180,E1 7300.594,E2 7300.594} C_VEL
LIN {X 0,Y 180.672,Z 985.024,A -85,B 0,C 180,E1 7296.355,E2 7296.355} C_VEL
LIN {X 0,Y 177.031,Z 993.364,A -85,B 0,C 180,E1 7291.619,E2 7291.619} C_VEL
LIN {X 0,Y 174.219,Z 1000.263,A -85,B 0,C 180,E1 7286.381,E2 7286.381} C_VEL
LIN {X 0,Y 172.426,Z 1005.684,A -85,B 0,C 180,E1 7280.657,E2 7280.657} C_VEL
LIN {X 0,Y 171.805,Z 1009.305,A -85,B 0,C 180,E1 7274.819,E2 7274.819} C_VEL
LIN {X 0,Y 172.34,Z 1011.134,A -85,B 0,C 180,E1 7268.919,E2 7268.919} C_VEL
LIN {X 0,Y 174.24,Z 1011.228,A -85,B 0,C 180,E1 7262.806,E2 7262.806} C_VEL
LIN {X 0,Y 177.577,Z 1009.486,A -85,B 0,C 180,E1 7256.897,E2 7256.897} C_VEL
LIN {X 0,Y 182.009,Z 1006.095,A -85,B 0,C 180,E1 7251.629,E2 7251.629} C_VEL
LIN {X 0,Y 187.746,Z 1000.866,A -85,B 0,C 180,E1 7246.608,E2 7246.608} C_VEL
LIN {X 0,Y 194.729,Z 993.636,A -85,B 0,C 180,E1 7241.875,E2 7241.875} C_VEL
LIN {X 0,Y 202.057,Z 985.057,A -85,B 0,C 180,E1 7237.851,E2 7237.851} C_VEL
LIN {X 0,Y 209.562,Z 975.011,A -85,B 0,C 180,E1 7234.37,E2 7234.37} C_VEL
LIN {X 0,Y 217.001,Z 963.642,A -85,B 0,C 180,E1 7231.377,E2 7231.377} C_VEL
LIN {X 0,Y 224.27,Z 950.81,A -85,B 0,C 180,E1 7228.784,E2 7228.784} C_VEL
LIN {X 0,Y 230.943,Z 936.927,A -85,B 0,C 180,E1 7226.617,E2 7226.617} C_VEL
LIN {X 0,Y 236.859,Z 922.001,A -85,B 0,C 180,E1 7224.828,E2 7224.828} C_VEL
LIN {X 0,Y 241.934,Z 905.783,A -85,B 0,C 180,E1 7223.351,E2 7223.351} C_VEL
LIN {X 0,Y 245.989,Z 888.332,A -85,B 0,C 180,E1 7222.176,E2 7222.176} C_VEL
LIN {X 0,Y 248.687,Z 870.769,A -85,B 0,C 180,E1 7221.349,E2 7221.349} C_VEL
LIN {X 0,Y 252.533,Z 827.24,A -85,B 0,C 180,E1 7220.163,E2 7220.163} C_VEL
LIN {X 0,Y 256.72,Z 779.655,A -85,B 0,C 180,E1 7218.979,E2 7218.979} C_VEL
LIN {X 0,Y 252.373,Z 770.323,A -85,B 0,C 180,E1 7216.042,E2 7216.042} C_VEL
LIN {X 0,Y 248.803,Z 763.224,A -85,B 0,C 180,E1 7213.242,E2 7213.242} C_VEL
LIN {X 0,Y 245.483,Z 757.362,A -85,B 0,C 180,E1 7210.206,E2 7210.206} C_VEL
LIN {X 0,Y 242.564,Z 752.183,A -85,B 0,C 180,E1 7206.747,E2 7206.747} C_VEL
LIN {X 0,Y 240.79,Z 749.314,A -85,B 0,C 180,E1 7204.007,E2 7204.007} C_VEL
LIN {X 0,Y 239.944,Z 748.52,A -85,B 0,C 180,E1 7202.454,E2 7202.454} C_VEL
LIN {X 0,Y 238.775,Z 749.704,A -85,B 0,C 180,E1 7200.221,E2 7200.221} C_VEL
LIN {X 0,Y 237.528,Z 752.973,A -85,B 0,C 180,E1 7196.477,E2 7196.477} C_VEL
LIN {X 0,Y 237.456,Z 753.211,A -85,B 0,C 180,E1 7195.519,E2 7195.519} C_VEL
LIN {X 0,Y 237.851,Z 753.854,A -85,B 0,C 180,E1 7191.783,E2 7191.783} C_VEL
LIN {X 0,Y 240.157,Z 757.554,A -85,B 0,C 180,E1 7186.273,E2 7186.273} C_VEL
LIN {X 0,Y 243.528,Z 763.402,A -85,B 0,C 180,E1 7181.695,E2 7181.695} C_VEL
LIN {X 0,Y 247.1,Z 770,A -85,B 0,C 180,E1 7178.207,E2 7178.207} C_VEL
LIN {X 0,Y 251.275,Z 778.269,A -85,B 0,C 180,E1 7174.864,E2 7174.864} C_VEL
LIN {X 0,Y 253.616,Z 783.707,A -85,B 0,C 180,E1 7173.193,E2 7173.193} C_VEL
LIN {X 0,Y 243.55,Z 893.083,A -85,B 0,C 180,E1 7170.541,E2 7170.541} C_VEL
LIN {X 0,Y 240.241,Z 911.7,A -85,B 0,C 180,E1 7169.855,E2 7169.855} C_VEL
LIN {X 0,Y 235.309,Z 930.281,A -85,B 0,C 180,E1 7168.892,E2 7168.892} C_VEL
LIN {X 0,Y 229.472,Z 946.984,A -85,B 0,C 180,E1 7167.703,E2 7167.703} C_VEL
LIN {X 0,Y 222.682,Z 962.927,A -85,B 0,C 180,E1 7166.166,E2 7166.166} C_VEL
LIN {X 0,Y 215.091,Z 978.104,A -85,B 0,C 180,E1 7164.209,E2 7164.209} C_VEL
LIN {X 0,Y 206.524,Z 993.02,A -85,B 0,C 180,E1 7161.655,E2 7161.655} C_VEL
LIN {X 0,Y 197.602,Z 1006.779,A -85,B 0,C 180,E1 7158.492,E2 7158.492} C_VEL
LIN {X 0,Y 188.913,Z 1019.002,A -85,B 0,C 180,E1 7154.742,E2 7154.742} C_VEL
LIN {X 0,Y 180.758,Z 1029.79,A -85,B 0,C 180,E1 7150.329,E2 7150.329} C_VEL
LIN {X 0,Y 173.286,Z 1039.475,A -85,B 0,C 180,E1 7144.982,E2 7144.982} C_VEL
LIN {X 0,Y 167.637,Z 1047.043,A -85,B 0,C 180,E1 7139.279,E2 7139.279} C_VEL
LIN {X 0,Y 163.692,Z 1053.047,A -85,B 0,C 180,E1 7133.011,E2 7133.011} C_VEL
LIN {X 0,Y 161.689,Z 1057.515,A -85,B 0,C 180,E1 7126.156,E2 7126.156} C_VEL
LIN {X 0,Y 161.705,Z 1060.111,A -85,B 0,C 180,E1 7119.25,E2 7119.25} C_VEL
LIN {X 0,Y 162.814,Z 1060.772,A -85,B 0,C 180,E1 7113.52,E2 7113.52} C_VEL
LIN {X 0,Y 163.393,Z 1060.361,A -85,B 0,C 180,E1 7109.648,E2 7109.648} C_VEL
LIN {X 0,Y 162.807,Z 1058.784,A -85,B 0,C 180,E1 7105.42,E2 7105.42} C_VEL
LIN {X 0,Y 162.309,Z 1057.609,A -85,B 0,C 180,E1 7102.566,E2 7102.566} C_VEL
LIN {X 0,Y 161.628,Z 1056.473,A -85,B 0,C 180,E1 7096.403,E2 7096.403} C_VEL
LIN {X 0,Y 162.682,Z 1053.398,A -85,B 0,C 180,E1 7089.867,E2 7089.867} C_VEL
LIN {X 0,Y 165.813,Z 1048.395,A -85,B 0,C 180,E1 7083.497,E2 7083.497} C_VEL
LIN {X 0,Y 171.383,Z 1041.073,A -85,B 0,C 180,E1 7077.14,E2 7077.14} C_VEL
LIN {X 0,Y 178.783,Z 1031.885,A -85,B 0,C 180,E1 7071.532,E2 7071.532} C_VEL
LIN {X 0,Y 187.269,Z 1021.461,A -85,B 0,C 180,E1 7066.888,E2 7066.888} C_VEL
LIN {X 0,Y 196.845,Z 1009.138,A -85,B 0,C 180,E1 7062.893,E2 7062.893} C_VEL
LIN {X 0,Y 206.542,Z 995.73,A -85,B 0,C 180,E1 7059.671,E2 7059.671} C_VEL
LIN {X 0,Y 216.177,Z 980.942,A -85,B 0,C 180,E1 7057.074,E2 7057.074} C_VEL
LIN {X 0,Y 224.944,Z 965.732,A -85,B 0,C 180,E1 7055.127,E2 7055.127} C_VEL
LIN {X 0,Y 232.98,Z 949.329,A -85,B 0,C 180,E1 7053.635,E2 7053.635} C_VEL
LIN {X 0,Y 239.274,Z 933.644,A -85,B 0,C 180,E1 7052.646,E2 7052.646} C_VEL
LIN {X 0,Y 245.184,Z 914.499,A -85,B 0,C 180,E1 7051.759,E2 7051.759} C_VEL
LIN {X 0,Y 252.299,Z 881.878,A -85,B 0,C 180,E1 7050.597,E2 7050.597} C_VEL
LIN {X 0,Y 246.813,Z 910.376,A -85,B 0,C 180,E1 7049.169,E2 7049.169} C_VEL
LIN {X 0,Y 242.944,Z 925.25,A -85,B 0,C 180,E1 7048.114,E2 7048.114} C_VEL
LIN {X 0,Y 237.393,Z 940.816,A -85,B 0,C 180,E1 7046.651,E2 7046.651} C_VEL
LIN {X 0,Y 231.101,Z 954.582,A -85,B 0,C 180,E1 7044.95,E2 7044.95} C_VEL
LIN {X 0,Y 223.866,Z 967.563,A -85,B 0,C 180,E1 7042.865,E2 7042.865} C_VEL
LIN {X 0,Y 215.196,Z 980.392,A -85,B 0,C 180,E1 7040.11,E2 7040.11} C_VEL
LIN {X 0,Y 206.91,Z 990.579,A -85,B 0,C 180,E1 7037.143,E2 7037.143} C_VEL
LIN {X 0,Y 199.161,Z 998.744,A -85,B 0,C 180,E1 7033.944,E2 7033.944} C_VEL
LIN {X 0,Y 191.465,Z 1005.549,A -85,B 0,C 180,E1 7030.227,E2 7030.227} C_VEL
LIN {X 0,Y 184.12,Z 1010.938,A -85,B 0,C 180,E1 7025.922,E2 7025.922} C_VEL
LIN {X 0,Y 177.397,Z 1014.594,A -85,B 0,C 180,E1 7020.968,E2 7020.968} C_VEL
LIN {X 0,Y 172.27,Z 1016.269,A -85,B 0,C 180,E1 7016.006,E2 7016.006} C_VEL
LIN {X 0,Y 168.084,Z 1016.137,A -85,B 0,C 180,E1 7010.411,E2 7010.411} C_VEL
LIN {X 0,Y 165.418,Z 1014.267,A -85,B 0,C 180,E1 7004.934,E2 7004.934} C_VEL
LIN {X 0,Y 163.877,Z 1010.288,A -85,B 0,C 180,E1 6998.989,E2 6998.989} C_VEL
LIN {X 0,Y 163.506,Z 1005.237,A -85,B 0,C 180,E1 6993.877,E2 6993.877} C_VEL
LIN {X 0,Y 164.027,Z 997.83,A -85,B 0,C 180,E1 6988.383,E2 6988.383} C_VEL
LIN {X 0,Y 165.298,Z 989.341,A -85,B 0,C 180,E1 6983.563,E2 6983.563} C_VEL
LIN {X 0,Y 167.327,Z 978.728,A -85,B 0,C 180,E1 6978.844,E2 6978.844} C_VEL
LIN {X 0,Y 169.755,Z 967.123,A -85,B 0,C 180,E1 6974.785,E2 6974.785} C_VEL
LIN {X 0,Y 172.527,Z 953.865,A -85,B 0,C 180,E1 6971.113,E2 6971.113} C_VEL
LIN {X 0,Y 175.421,Z 938.903,A -85,B 0,C 180,E1 6967.894,E2 6967.894} C_VEL
LIN {X 0,Y 177.971,Z 923.714,A -85,B 0,C 180,E1 6965.358,E2 6965.358} C_VEL
LIN {X 0,Y 180.137,Z 909.705,A -85,B 0,C 180,E1 6963.395,E2 6963.395} C_VEL
LIN {X 0,Y 180.975,Z 908.54,A -85,B 0,C 180,E1 6962.882,E2 6962.882} C_VEL
LIN {X 0,Y 183.08,Z 907.941,A -85,B 0,C 180,E1 6962.165,E2 6962.165} C_VEL
LIN {X 0,Y 185.554,Z 906.185,A -85,B 0,C 180,E1 6961.636,E2 6961.636} C_VEL
LIN {X 0,Y 189.258,Z 901.954,A -85,B 0,C 180,E1 6961.144,E2 6961.144} C_VEL
LIN {X 0,Y 190.738,Z 899.845,A -85,B 0,C 180,E1 6961.009,E2 6961.009} C_VEL
LIN {X 0,Y 194.337,Z 897.813,A -85,B 0,C 180,E1 6960.189,E2 6960.189} C_VEL
LIN {X 0,Y 198.287,Z 893.788,A -85,B 0,C 180,E1 6959.56,E2 6959.56} C_VEL
LIN {X 0,Y 202.393,Z 887.495,A -85,B 0,C 180,E1 6959.168,E2 6959.168} C_VEL
LIN {X 0,Y 204.958,Z 882.423,A -85,B 0,C 180,E1 6959.019,E2 6959.019} C_VEL
LIN {X 0,Y 206.414,Z 881.25,A -85,B 0,C 180,E1 6958.728,E2 6958.728} C_VEL
LIN {X 0,Y 203.752,Z 897.687,A -85,B 0,C 180,E1 6957.471,E2 6957.471} C_VEL
LIN {X 0,Y 200.147,Z 913.88,A -85,B 0,C 180,E1 6955.762,E2 6955.762} C_VEL
LIN {X 0,Y 195.633,Z 930.032,A -85,B 0,C 180,E1 6953.495,E2 6953.495} C_VEL
LIN {X 0,Y 190.621,Z 945.054,A -85,B 0,C 180,E1 6950.736,E2 6950.736} C_VEL
LIN {X 0,Y 185.308,Z 958.813,A -85,B 0,C 180,E1 6947.426,E2 6947.426} C_VEL
LIN {X 0,Y 179.93,Z 971.423,A -85,B 0,C 180,E1 6943.498,E2 6943.498} C_VEL
LIN {X 0,Y 175.097,Z 982.081,A -85,B 0,C 180,E1 6939.201,E2 6939.201} C_VEL
LIN {X 0,Y 170.84,Z 991.234,A -85,B 0,C 180,E1 6934.364,E2 6934.364} C_VEL
LIN {X 0,Y 167.42,Z 998.91,A -85,B 0,C 180,E1 6928.974,E2 6928.974} C_VEL
LIN {X 0,Y 165.067,Z 1005.071,A -85,B 0,C 180,E1 6923.043,E2 6923.043} C_VEL
LIN {X 0,Y 163.972,Z 1009.338,A -85,B 0,C 180,E1 6916.962,E2 6916.962} C_VEL
LIN {X 0,Y 164.113,Z 1011.827,A -85,B 0,C 180,E1 6910.793,E2 6910.793} C_VEL
LIN {X 0,Y 165.565,Z 1012.627,A -85,B 0,C 180,E1 6904.611,E2 6904.611} C_VEL
LIN {X 0,Y 168.455,Z 1011.702,A -85,B 0,C 180,E1 6898.513,E2 6898.513} C_VEL
LIN {X 0,Y 172.873,Z 1008.905,A -85,B 0,C 180,E1 6892.607,E2 6892.607} C_VEL
LIN {X 0,Y 178.635,Z 1004.305,A -85,B 0,C 180,E1 6887.159,E2 6887.159} C_VEL
LIN {X 0,Y 185.322,Z 998.134,A -85,B 0,C 180,E1 6882.342,E2 6882.342} C_VEL
LIN {X 0,Y 192.856,Z 990.238,A -85,B 0,C 180,E1 6877.998,E2 6877.998} C_VEL
LIN {X 0,Y 200.727,Z 980.761,A -85,B 0,C 180,E1 6874.222,E2 6874.222} C_VEL
LIN {X 0,Y 208.695,Z 969.8,A -85,B 0,C 180,E1 6870.954,E2 6870.954} C_VEL
LIN {X 0,Y 216.555,Z 957.325,A -85,B 0,C 180,E1 6868.133,E2 6868.133} C_VEL
LIN {X 0,Y 223.78,Z 943.879,A -85,B 0,C 180,E1 6865.802,E2 6865.802} C_VEL
LIN {X 0,Y 230.228,Z 929.411,A -85,B 0,C 180,E1 6863.881,E2 6863.881} C_VEL
LIN {X 0,Y 235.666,Z 914.404,A -85,B 0,C 180,E1 6862.347,E2 6862.347} C_VEL
LIN {X 0,Y 240.47,Z 897.202,A -85,B 0,C 180,E1 6861.021,E2 6861.021} C_VEL
LIN {X 0,Y 243.859,Z 880.013,A -85,B 0,C 180,E1 6860.064,E2 6860.064} C_VEL
LIN {X 0,Y 245.951,Z 861.951,A -85,B 0,C 180,E1 6859.393,E2 6859.393} C_VEL
LIN {X 0,Y 253.111,Z 783.937,A -85,B 0,C 180,E1 6857.471,E2 6857.471} C_VEL
LIN {X 0,Y 249.048,Z 774.781,A -85,B 0,C 180,E1 6854.414,E2 6854.414} C_VEL
LIN {X 0,Y 245.507,Z 767.945,A -85,B 0,C 180,E1 6851.333,E2 6851.333} C_VEL
LIN {X 0,Y 242.589,Z 762.375,A -85,B 0,C 180,E1 6848.175,E2 6848.175} C_VEL
LIN {X 0,Y 240.856,Z 759.4,A -85,B 0,C 180,E1 6845.838,E2 6845.838} C_VEL
LIN {X 0,Y 238.967,Z 755.859,A -85,B 0,C 180,E1 6842.398,E2 6842.398} C_VEL
LIN {X 0,Y 237.524,Z 753.276,A -85,B 0,C 180,E1 6836.863,E2 6836.863} C_VEL
LIN {X 0,Y 237.456,Z 753.211,A -85,B 0,C 180,E1 6835.519,E2 6835.519} C_VEL
LIN {X 0,Y 237.421,Z 754.273,A -85,B 0,C 180,E1 6833.802,E2 6833.802} C_VEL
LIN {X 0,Y 237.438,Z 758.187,A -85,B 0,C 180,E1 6831.418,E2 6831.418} C_VEL
LIN {X 0,Y 237.992,Z 763.366,A -85,B 0,C 180,E1 6828.538,E2 6828.538} C_VEL
LIN {X 0,Y 238.521,Z 764.587,A -85,B 0,C 180,E1 6827.362,E2 6827.362} C_VEL
LIN {X 0,Y 241.883,Z 770.783,A -85,B 0,C 180,E1 6822.313,E2 6822.313} C_VEL
LIN {X 0,Y 245.295,Z 777.403,A -85,B 0,C 180,E1 6818.792,E2 6818.792} C_VEL
LIN {X 0,Y 249.09,Z 785.373,A -85,B 0,C 180,E1 6815.579,E2 6815.579} C_VEL
LIN {X 0,Y 250.104,Z 787.986,A -85,B 0,C 180,E1 6814.775,E2 6814.775} C_VEL
LIN {X 0,Y 240.115,Z 892.432,A -85,B 0,C 180,E1 6812.266,E2 6812.266} C_VEL
LIN {X 0,Y 236.719,Z 910.98,A -85,B 0,C 180,E1 6811.595,E2 6811.595} C_VEL
LIN {X 0,Y 231.685,Z 929.438,A -85,B 0,C 180,E1 6810.662,E2 6810.662} C_VEL
LIN {X 0,Y 225.69,Z 946.123,A -85,B 0,C 180,E1 6809.504,E2 6809.504} C_VEL
LIN {X 0,Y 218.693,Z 962.044,A -85,B 0,C 180,E1 6808.005,E2 6808.005} C_VEL
LIN {X 0,Y 210.841,Z 977.197,A -85,B 0,C 180,E1 6806.086,E2 6806.086} C_VEL
LIN {X 0,Y 202.289,Z 991.526,A -85,B 0,C 180,E1 6803.673,E2 6803.673} C_VEL
LIN {X 0,Y 192.944,Z 1005.367,A -85,B 0,C 180,E1 6800.545,E2 6800.545} C_VEL
LIN {X 0,Y 183.776,Z 1017.628,A -85,B 0,C 180,E1 6796.806,E2 6796.806} C_VEL
LIN {X 0,Y 175.084,Z 1028.436,A -85,B 0,C 180,E1 6792.365,E2 6792.365} C_VEL
LIN {X 0,Y 166.868,Z 1038.295,A -85,B 0,C 180,E1 6786.811,E2 6786.811} C_VEL
LIN {X 0,Y 160.506,Z 1046.094,A -85,B 0,C 180,E1 6780.717,E2 6780.717} C_VEL
LIN {X 0,Y 155.971,Z 1052.316,A -85,B 0,C 180,E1 6773.819,E2 6773.819} C_VEL
LIN {X 0,Y 153.783,Z 1056.573,A -85,B 0,C 180,E1 6766.622,E2 6766.622} C_VEL
LIN {X 0,Y 153.756,Z 1058.973,A -85,B 0,C 180,E1 6759.355,E2 6759.355} C_VEL
LIN {X 0,Y 154.925,Z 1059.547,A -85,B 0,C 180,E1 6753.329,E2 6753.329} C_VEL
LIN {X 0,Y 155.494,Z 1059.062,A -85,B 0,C 180,E1 6749.631,E2 6749.631} C_VEL
LIN {X 0,Y 154.831,Z 1057.418,A -85,B 0,C 180,E1 6745.183,E2 6745.183} C_VEL
LIN {X 0,Y 154.345,Z 1056.099,A -85,B 0,C 180,E1 6742.18,E2 6742.18} C_VEL
LIN {X 0,Y 153.712,Z 1055.24,A -85,B 0,C 180,E1 6735.688,E2 6735.688} C_VEL
LIN {X 0,Y 154.992,Z 1052.406,A -85,B 0,C 180,E1 6728.821,E2 6728.821} C_VEL
LIN {X 0,Y 158.761,Z 1047.489,A -85,B 0,C 180,E1 6721.812,E2 6721.812} C_VEL
LIN {X 0,Y 164.567,Z 1040.885,A -85,B 0,C 180,E1 6715.594,E2 6715.594} C_VEL
LIN {X 0,Y 172.413,Z 1032.401,A -85,B 0,C 180,E1 6709.93,E2 6709.93} C_VEL
LIN {X 0,Y 181.534,Z 1022.422,A -85,B 0,C 180,E1 6705.169,E2 6705.169} C_VEL
LIN {X 0,Y 192.126,Z 1010.298,A -85,B 0,C 180,E1 6701.008,E2 6701.008} C_VEL
LIN {X 0,Y 202.461,Z 997.376,A -85,B 0,C 180,E1 6697.798,E2 6697.798} C_VEL
LIN {X 0,Y 212.909,Z 982.968,A -85,B 0,C 180,E1 6695.2,E2 6695.2} C_VEL
LIN {X 0,Y 222.79,Z 967.337,A -85,B 0,C 180,E1 6693.197,E2 6693.197} C_VEL
LIN {X 0,Y 231.176,Z 951.878,A -85,B 0,C 180,E1 6691.8,E2 6691.8} C_VEL
LIN {X 0,Y 238.115,Z 936.276,A -85,B 0,C 180,E1 6690.827,E2 6690.827} C_VEL
LIN {X 0,Y 242.804,Z 923.464,A -85,B 0,C 180,E1 6690.211,E2 6690.211} C_VEL
LIN {X 0,Y 237.578,Z 938.298,A -85,B 0,C 180,E1 6688.945,E2 6688.945} C_VEL
LIN {X 0,Y 230.962,Z 952.872,A -85,B 0,C 180,E1 6687.315,E2 6687.315} C_VEL
LIN {X 0,Y 223.269,Z 966.395,A -85,B 0,C 180,E1 6685.32,E2 6685.32} C_VEL
LIN {X 0,Y 215.036,Z 978.401,A -85,B 0,C 180,E1 6682.977,E2 6682.977} C_VEL
LIN {X 0,Y 206.13,Z 989.23,A -85,B 0,C 180,E1 6680.144,E2 6680.144} C_VEL
LIN {X 0,Y 197.674,Z 997.936,A -85,B 0,C 180,E1 6677.059,E2 6677.059} C_VEL
LIN {X 0,Y 188.625,Z 1005.751,A -85,B 0,C 180,E1 6673.175,E2 6673.175} C_VEL
LIN {X 0,Y 180.44,Z 1011.461,A -85,B 0,C 180,E1 6668.925,E2 6668.925} C_VEL
LIN {X 0,Y 173.284,Z 1015.347,A -85,B 0,C 180,E1 6664.301,E2 6664.301} C_VEL
LIN {X 0,Y 166.888,Z 1017.518,A -85,B 0,C 180,E1 6658.969,E2 6658.969} C_VEL
LIN {X 0,Y 161.896,Z 1017.824,A -85,B 0,C 180,E1 6653.261,E2 6653.261} C_VEL
LIN {X 0,Y 158.344,Z 1016.139,A -85,B 0,C 180,E1 6647.231,E2 6647.231} C_VEL
LIN {X 0,Y 156.348,Z 1012.75,A -85,B 0,C 180,E1 6641.351,E2 6641.351} C_VEL
LIN {X 0,Y 155.546,Z 1007.376,A -85,B 0,C 180,E1 6635.302,E2 6635.302} C_VEL
LIN {X 0,Y 155.782,Z 1000.867,A -85,B 0,C 180,E1 6629.958,E2 6629.958} C_VEL
LIN {X 0,Y 156.929,Z 992.266,A -85,B 0,C 180,E1 6624.563,E2 6624.563} C_VEL
LIN {X 0,Y 158.653,Z 983.029,A -85,B 0,C 180,E1 6619.997,E2 6619.997} C_VEL
LIN {X 0,Y 161.238,Z 970.82,A -85,B 0,C 180,E1 6615.264,E2 6615.264} C_VEL
LIN {X 0,Y 164.075,Z 957.731,A -85,B 0,C 180,E1 6611.3,E2 6611.3} C_VEL
LIN {X 0,Y 166.909,Z 944.057,A -85,B 0,C 180,E1 6608.024,E2 6608.024} C_VEL
LIN {X 0,Y 169.814,Z 928.124,A -85,B 0,C 180,E1 6605.071,E2 6605.071} C_VEL
LIN {X 0,Y 170.972,Z 922.124,A -85,B 0,C 180,E1 6604.006,E2 6604.006} C_VEL
LIN {X 0,Y 171.604,Z 921.247,A -85,B 0,C 180,E1 6603.57,E2 6603.57} C_VEL
LIN {X 0,Y 174.381,Z 920.541,A -85,B 0,C 180,E1 6602.555,E2 6602.555} C_VEL
LIN {X 0,Y 177.754,Z 918.19,A -85,B 0,C 180,E1 6601.855,E2 6601.855} C_VEL
LIN {X 0,Y 180.546,Z 915.511,A -85,B 0,C 180,E1 6601.476,E2 6601.476} C_VEL
LIN {X 0,Y 184.464,Z 913.86,A -85,B 0,C 180,E1 6600.475,E2 6600.475} C_VEL
LIN {X 0,Y 188.853,Z 910.357,A -85,B 0,C 180,E1 6599.739,E2 6599.739} C_VEL
LIN {X 0,Y 193.136,Z 905.689,A -85,B 0,C 180,E1 6599.269,E2 6599.269} C_VEL
LIN {X 0,Y 196.893,Z 903.225,A -85,B 0,C 180,E1 6598.555,E2 6598.555} C_VEL
LIN {X 0,Y 192.825,Z 919.656,A -85,B 0,C 180,E1 6596.65,E2 6596.65} C_VEL
LIN {X 0,Y 188.153,Z 934.764,A -85,B 0,C 180,E1 6594.322,E2 6594.322} C_VEL
LIN {X 0,Y 182.749,Z 949.596,A -85,B 0,C 180,E1 6591.337,E2 6591.337} C_VEL
LIN {X 0,Y 177.304,Z 962.769,A -85,B 0,C 180,E1 6587.9,E2 6587.9} C_VEL
LIN {X 0,Y 172.171,Z 974.074,A -85,B 0,C 180,E1 6584.107,E2 6584.107} C_VEL
LIN {X 0,Y 167.196,Z 984.361,A -85,B 0,C 180,E1 6579.64,E2 6579.64} C_VEL
LIN {X 0,Y 162.83,Z 993.284,A -85,B 0,C 180,E1 6574.58,E2 6574.58} C_VEL
LIN {X 0,Y 159.35,Z 1000.779,A -85,B 0,C 180,E1 6568.922,E2 6568.922} C_VEL
LIN {X 0,Y 157.109,Z 1006.454,A -85,B 0,C 180,E1 6563.056,E2 6563.056} C_VEL
LIN {X 0,Y 156.02,Z 1010.637,A -85,B 0,C 180,E1 6556.662,E2 6556.662} C_VEL
LIN {X 0,Y 156.271,Z 1013.089,A -85,B 0,C 180,E1 6550.145,E2 6550.145} C_VEL
LIN {X 0,Y 157.926,Z 1013.841,A -85,B 0,C 180,E1 6543.694,E2 6543.694} C_VEL
LIN {X 0,Y 161.126,Z 1012.88,A -85,B 0,C 180,E1 6537.326,E2 6537.326} C_VEL
LIN {X 0,Y 165.94,Z 1010.031,A -85,B 0,C 180,E1 6531.198,E2 6531.198} C_VEL
LIN {X 0,Y 172.122,Z 1005.413,A -85,B 0,C 180,E1 6525.604,E2 6525.604} C_VEL
LIN {X 0,Y 179.27,Z 999.199,A -85,B 0,C 180,E1 6520.667,E2 6520.667} C_VEL
LIN {X 0,Y 187.238,Z 991.268,A -85,B 0,C 180,E1 6516.261,E2 6516.261} C_VEL
LIN {X 0,Y 195.512,Z 981.76,A -85,B 0,C 180,E1 6512.456,E2 6512.456} C_VEL
LIN {X 0,Y 203.848,Z 970.781,A -85,B 0,C 180,E1 6509.183,E2 6509.183} C_VEL
LIN {X 0,Y 212.036,Z 958.289,A -85,B 0,C 180,E1 6506.371,E2 6506.371} C_VEL
LIN {X 0,Y 219.539,Z 944.828,A -85,B 0,C 180,E1 6504.057,E2 6504.057} C_VEL
LIN {X 0,Y 226.182,Z 930.443,A -85,B 0,C 180,E1 6502.165,E2 6502.165} C_VEL
LIN {X 0,Y 231.848,Z 915.393,A -85,B 0,C 180,E1 6500.64,E2 6500.64} C_VEL
LIN {X 0,Y 236.818,Z 898.279,A -85,B 0,C 180,E1 6499.332,E2 6499.332} C_VEL
LIN {X 0,Y 240.352,Z 881.108,A -85,B 0,C 180,E1 6498.38,E2 6498.38} C_VEL
LIN {X 0,Y 242.557,Z 863.139,A -85,B 0,C 180,E1 6497.712,E2 6497.712} C_VEL
LIN {X 0,Y 249.642,Z 788.184,A -85,B 0,C 180,E1 6495.87,E2 6495.87} C_VEL
LIN {X 0,Y 246.194,Z 780.336,A -85,B 0,C 180,E1 6493.027,E2 6493.027} C_VEL
LIN {X 0,Y 243.12,Z 774.018,A -85,B 0,C 180,E1 6490.067,E2 6490.067} C_VEL
LIN {X 0,Y 239.992,Z 767.739,A -85,B 0,C 180,E1 6486.099,E2 6486.099} C_VEL
LIN {X 0,Y 237.729,Z 763.582,A -85,B 0,C 180,E1 6481.929,E2 6481.929} C_VEL
LIN {X 0,Y 236.495,Z 761.19,A -85,B 0,C 180,E1 6476.607,E2 6476.607} C_VEL
LIN {X 0,Y 236.753,Z 761.622,A -85,B 0,C 180,E1 6472.234,E2 6472.234} C_VEL
LIN {X 0,Y 238.521,Z 764.587,A -85,B 0,C 180,E1 6467.362,E2 6467.362} C_VEL
LIN {X 0,Y 239.292,Z 766.603,A -85,B 0,C 180,E1 6465.861,E2 6465.861} C_VEL
LIN {X 0,Y 240.161,Z 771.266,A -85,B 0,C 180,E1 6464.055,E2 6464.055} C_VEL
LIN {X 0,Y 242.14,Z 781.53,A -85,B 0,C 180,E1 6460.837,E2 6460.837} C_VEL
LIN {X 0,Y 242.758,Z 783.196,A -85,B 0,C 180,E1 6460.146,E2 6460.146} C_VEL
LIN {X 0,Y 246.55,Z 791.451,A -85,B 0,C 180,E1 6456.646,E2 6456.646} C_VEL
LIN {X 0,Y 246.799,Z 792.494,A -85,B 0,C 180,E1 6456.397,E2 6456.397} C_VEL
LIN {X 0,Y 236.985,Z 891.577,A -85,B 0,C 180,E1 6454.051,E2 6454.051} C_VEL
LIN {X 0,Y 233.501,Z 910.068,A -85,B 0,C 180,E1 6453.397,E2 6453.397} C_VEL
LIN {X 0,Y 228.29,Z 928.644,A -85,B 0,C 180,E1 6452.486,E2 6452.486} C_VEL
LIN {X 0,Y 222.14,Z 945.261,A -85,B 0,C 180,E1 6451.365,E2 6451.365} C_VEL
LIN {X 0,Y 214.939,Z 961.162,A -85,B 0,C 180,E1 6449.909,E2 6449.909} C_VEL
LIN {X 0,Y 206.829,Z 976.291,A -85,B 0,C 180,E1 6448.038,E2 6448.038} C_VEL
LIN {X 0,Y 197.601,Z 991.139,A -85,B 0,C 180,E1 6445.565,E2 6445.565} C_VEL
LIN {X 0,Y 187.878,Z 1004.823,A -85,B 0,C 180,E1 6442.461,E2 6442.461} C_VEL
LIN {X 0,Y 178.282,Z 1016.982,A -85,B 0,C 180,E1 6438.72,E2 6438.72} C_VEL
LIN {X 0,Y 169.114,Z 1027.694,A -85,B 0,C 180,E1 6434.238,E2 6434.238} C_VEL
LIN {X 0,Y 160.798,Z 1036.969,A -85,B 0,C 180,E1 6428.904,E2 6428.904} C_VEL
LIN {X 0,Y 153.812,Z 1044.765,A -85,B 0,C 180,E1 6422.651,E2 6422.651} C_VEL
LIN {X 0,Y 148.687,Z 1050.996,A -85,B 0,C 180,E1 6415.49,E2 6415.49} C_VEL
LIN {X 0,Y 146.009,Z 1055.31,A -85,B 0,C 180,E1 6407.852,E2 6407.852} C_VEL
LIN {X 0,Y 145.713,Z 1057.696,A -85,B 0,C 180,E1 6400.276,E2 6400.276} C_VEL
LIN {X 0,Y 146.951,Z 1058.279,A -85,B 0,C 180,E1 6393.51,E2 6393.51} C_VEL
LIN {X 0,Y 147.593,Z 1057.758,A -85,B 0,C 180,E1 6389.611,E2 6389.611} C_VEL
LIN {X 0,Y 146.849,Z 1056.052,A -85,B 0,C 180,E1 6384.921,E2 6384.921} C_VEL
LIN {X 0,Y 146.31,Z 1054.543,A -85,B 0,C 180,E1 6381.352,E2 6381.352} C_VEL
LIN {X 0,Y 145.889,Z 1053.719,A -85,B 0,C 180,E1 6374.088,E2 6374.088} C_VEL
LIN {X 0,Y 147.674,Z 1051.019,A -85,B 0,C 180,E1 6366.876,E2 6366.876} C_VEL
LIN {X 0,Y 152.168,Z 1046.24,A -85,B 0,C 180,E1 6359.605,E2 6359.605} C_VEL
LIN {X 0,Y 158.72,Z 1039.921,A -85,B 0,C 180,E1 6353.24,E2 6353.24} C_VEL
LIN {X 0,Y 167.355,Z 1031.709,A -85,B 0,C 180,E1 6347.535,E2 6347.535} C_VEL
LIN {X 0,Y 177.842,Z 1021.535,A -85,B 0,C 180,E1 6342.564,E2 6342.564} C_VEL
LIN {X 0,Y 189.176,Z 1009.726,A -85,B 0,C 180,E1 6338.534,E2 6338.534} C_VEL
LIN {X 0,Y 200.121,Z 997.288,A -85,B 0,C 180,E1 6335.471,E2 6335.471} C_VEL
LIN {X 0,Y 211.078,Z 983.329,A -85,B 0,C 180,E1 6333.023,E2 6333.023} C_VEL
LIN {X 0,Y 221.422,Z 968.345,A -85,B 0,C 180,E1 6331.16,E2 6331.16} C_VEL
LIN {X 0,Y 230.499,Z 952.81,A -85,B 0,C 180,E1 6329.822,E2 6329.822} C_VEL
LIN {X 0,Y 231.457,Z 951.037,A -85,B 0,C 180,E1 6329.678,E2 6329.678} C_VEL
LIN {X 0,Y 223.257,Z 965.357,A -85,B 0,C 180,E1 6327.759,E2 6327.759} C_VEL
LIN {X 0,Y 214.89,Z 977.249,A -85,B 0,C 180,E1 6325.64,E2 6325.64} C_VEL
LIN {X 0,Y 206.085,Z 987.872,A -85,B 0,C 180,E1 6323.14,E2 6323.14} C_VEL
LIN {X 0,Y 196.237,Z 997.739,A -85,B 0,C 180,E1 6319.96,E2 6319.96} C_VEL
LIN {X 0,Y 187.018,Z 1005.467,A -85,B 0,C 180,E1 6316.46,E2 6316.46} C_VEL
LIN {X 0,Y 177.376,Z 1012.032,A -85,B 0,C 180,E1 6312.038,E2 6312.038} C_VEL
LIN {X 0,Y 168.844,Z 1016.424,A -85,B 0,C 180,E1 6307.143,E2 6307.143} C_VEL
LIN {X 0,Y 161.617,Z 1018.868,A -85,B 0,C 180,E1 6301.772,E2 6301.772} C_VEL
LIN {X 0,Y 155.812,Z 1019.369,A -85,B 0,C 180,E1 6295.952,E2 6295.952} C_VEL
LIN {X 0,Y 151.757,Z 1018.147,A -85,B 0,C 180,E1 6290.136,E2 6290.136} C_VEL
LIN {X 0,Y 148.951,Z 1014.867,A -85,B 0,C 180,E1 6283.624,E2 6283.624} C_VEL
LIN {X 0,Y 147.742,Z 1010.278,A -85,B 0,C 180,E1 6277.728,E2 6277.728} C_VEL
LIN {X 0,Y 147.617,Z 1003.731,A -85,B 0,C 180,E1 6271.696,E2 6271.696} C_VEL
LIN {X 0,Y 148.498,Z 995.658,A -85,B 0,C 180,E1 6266.023,E2 6266.023} C_VEL
LIN {X 0,Y 150.398,Z 985.11,A -85,B 0,C 180,E1 6260.34,E2 6260.34} C_VEL
LIN {X 0,Y 152.915,Z 973.4,A -85,B 0,C 180,E1 6255.458,E2 6255.458} C_VEL
LIN {X 0,Y 155.758,Z 960.821,A -85,B 0,C 180,E1 6251.316,E2 6251.316} C_VEL
LIN {X 0,Y 158.926,Z 946.162,A -85,B 0,C 180,E1 6247.559,E2 6247.559} C_VEL
LIN {X 0,Y 161.7,Z 932.868,A -85,B 0,C 180,E1 6244.731,E2 6244.731} C_VEL
LIN {X 0,Y 162.506,Z 932.093,A -85,B 0,C 180,E1 6244.151,E2 6244.151} C_VEL
LIN {X 0,Y 164.902,Z 931.653,A -85,B 0,C 180,E1 6243.201,E2 6243.201} C_VEL
LIN {X 0,Y 168.194,Z 929.766,A -85,B 0,C 180,E1 6242.418,E2 6242.418} C_VEL
LIN {X 0,Y 170.424,Z 928.087,A -85,B 0,C 180,E1 6242.029,E2 6242.029} C_VEL
LIN {X 0,Y 173.85,Z 927.026,A -85,B 0,C 180,E1 6241.024,E2 6241.024} C_VEL
LIN {X 0,Y 178.104,Z 924.412,A -85,B 0,C 180,E1 6240.168,E2 6240.168} C_VEL
LIN {X 0,Y 181.33,Z 921.808,A -85,B 0,C 180,E1 6239.719,E2 6239.719} C_VEL
LIN {X 0,Y 185.913,Z 919.508,A -85,B 0,C 180,E1 6238.76,E2 6238.76} C_VEL
LIN {X 0,Y 187.369,Z 918.694,A -85,B 0,C 180,E1 6238.477,E2 6238.477} C_VEL
LIN {X 0,Y 182.556,Z 934.016,A -85,B 0,C 180,E1 6236.162,E2 6236.162} C_VEL
LIN {X 0,Y 177.108,Z 948.551,A -85,B 0,C 180,E1 6233.278,E2 6233.278} C_VEL
LIN {X 0,Y 171.325,Z 962.062,A -85,B 0,C 180,E1 6229.786,E2 6229.786} C_VEL
LIN {X 0,Y 165.656,Z 974.061,A -85,B 0,C 180,E1 6225.761,E2 6225.761} C_VEL
LIN {X 0,Y 160.329,Z 984.629,A -85,B 0,C 180,E1 6221.148,E2 6221.148} C_VEL
LIN {X 0,Y 155.622,Z 993.713,A -85,B 0,C 180,E1 6215.901,E2 6215.901} C_VEL
LIN {X 0,Y 151.838,Z 1001.354,A -85,B 0,C 180,E1 6210.001,E2 6210.001} C_VEL
LIN {X 0,Y 149.362,Z 1007.17,A -85,B 0,C 180,E1 6203.852,E2 6203.852} C_VEL
LIN {X 0,Y 148.127,Z 1011.56,A -85,B 0,C 180,E1 6197.13,E2 6197.13} C_VEL
LIN {X 0,Y 148.318,Z 1014.146,A -85,B 0,C 180,E1 6190.303,E2 6190.303} C_VEL
LIN {X 0,Y 150.135,Z 1015.051,A -85,B 0,C 180,E1 6183.178,E2 6183.178} C_VEL
LIN {X 0,Y 153.616,Z 1014.151,A -85,B 0,C 180,E1 6176.411,E2 6176.411} C_VEL
LIN {X 0,Y 158.762,Z 1011.391,A -85,B 0,C 180,E1 6170.032,E2 6170.032} C_VEL
LIN {X 0,Y 165.127,Z 1006.993,A -85,B 0,C 180,E1 6164.399,E2 6164.399} C_VEL
LIN {X 0,Y 172.857,Z 1000.711,A -85,B 0,C 180,E1 6159.187,E2 6159.187} C_VEL
LIN {X 0,Y 181.212,Z 992.886,A -85,B 0,C 180,E1 6154.703,E2 6154.703} C_VEL
LIN {X 0,Y 189.852,Z 983.536,A -85,B 0,C 180,E1 6150.859,E2 6150.859} C_VEL
LIN {X 0,Y 198.517,Z 972.7,A -85,B 0,C 180,E1 6147.571,E2 6147.571} C_VEL
LIN {X 0,Y 207.365,Z 959.845,A -85,B 0,C 180,E1 6144.648,E2 6144.648} C_VEL
LIN {X 0,Y 215.136,Z 946.534,A -85,B 0,C 180,E1 6142.353,E2 6142.353} C_VEL
LIN {X 0,Y 222.009,Z 932.432,A -85,B 0,C 180,E1 6140.486,E2 6140.486} C_VEL
LIN {X 0,Y 228.25,Z 916.506,A -85,B 0,C 180,E1 6138.882,E2 6138.882} C_VEL
LIN {X 0,Y 233.384,Z 899.461,A -85,B 0,C 180,E1 6137.594,E2 6137.594} C_VEL
LIN {X 0,Y 237.072,Z 882.233,A -85,B 0,C 180,E1 6136.648,E2 6136.648} C_VEL
LIN {X 0,Y 239.387,Z 864.294,A -85,B 0,C 180,E1 6135.983,E2 6135.983} C_VEL
LIN {X 0,Y 246.358,Z 792.422,A -85,B 0,C 180,E1 6134.214,E2 6134.214} C_VEL
LIN {X 0,Y 243.045,Z 784.725,A -85,B 0,C 180,E1 6131.149,E2 6131.149} C_VEL
LIN {X 0,Y 240.27,Z 778.962,A -85,B 0,C 180,E1 6128.014,E2 6128.014} C_VEL
LIN {X 0,Y 238.403,Z 775.073,A -85,B 0,C 180,E1 6125.295,E2 6125.295} C_VEL
LIN {X 0,Y 236.507,Z 771.308,A -85,B 0,C 180,E1 6121.454,E2 6121.454} C_VEL
LIN {X 0,Y 235.47,Z 769.11,A -85,B 0,C 180,E1 6116.349,E2 6116.349} C_VEL
LIN {X 0,Y 235.744,Z 769.621,A -85,B 0,C 180,E1 6112.2,E2 6112.2} C_VEL
LIN {X 0,Y 237.602,Z 772.984,A -85,B 0,C 180,E1 6107.113,E2 6107.113} C_VEL
LIN {X 0,Y 240.522,Z 778.626,A -85,B 0,C 180,E1 6102.647,E2 6102.647} C_VEL
LIN {X 0,Y 242.758,Z 783.196,A -85,B 0,C 180,E1 6100.146,E2 6100.146} C_VEL
LIN {X 0,Y 243.42,Z 785.801,A -85,B 0,C 180,E1 6099.358,E2 6099.358} C_VEL
LIN {X 0,Y 243.777,Z 790.31,A -85,B 0,C 180,E1 6098.646,E2 6098.646} C_VEL
LIN {X 0,Y 243.662,Z 796.622,A -85,B 0,C 180,E1 6098.124,E2 6098.124} C_VEL
LIN {X 0,Y 242.581,Z 808.581,A -85,B 0,C 180,E1 6097.761,E2 6097.761} C_VEL
LIN {X 0,Y 241.654,Z 817.078,A -85,B 0,C 180,E1 6097.614,E2 6097.614} C_VEL
LIN {X 0,Y 234.095,Z 890.877,A -85,B 0,C 180,E1 6095.879,E2 6095.879} C_VEL
LIN {X 0,Y 230.498,Z 909.424,A -85,B 0,C 180,E1 6095.242,E2 6095.242} C_VEL
LIN {X 0,Y 225.138,Z 928.016,A -85,B 0,C 180,E1 6094.36,E2 6094.36} C_VEL
LIN {X 0,Y 218.836,Z 944.565,A -85,B 0,C 180,E1 6093.282,E2 6093.282} C_VEL
LIN {X 0,Y 211.031,Z 961.188,A -85,B 0,C 180,E1 6091.794,E2 6091.794} C_VEL
LIN {X 0,Y 202.288,Z 976.731,A -85,B 0,C 180,E1 6089.879,E2 6089.879} C_VEL
LIN {X 0,Y 192.765,Z 991.229,A -85,B 0,C 180,E1 6087.444,E2 6087.444} C_VEL
LIN {X 0,Y 183.034,Z 1004.281,A -85,B 0,C 180,E1 6084.482,E2 6084.482} C_VEL
LIN {X 0,Y 173.001,Z 1016.338,A -85,B 0,C 180,E1 6080.754,E2 6080.754} C_VEL
LIN {X 0,Y 163.297,Z 1027.003,A -85,B 0,C 180,E1 6076.221,E2 6076.221} C_VEL
LIN {X 0,Y 154.343,Z 1036.287,A -85,B 0,C 180,E1 6070.718,E2 6070.718} C_VEL
LIN {X 0,Y 146.945,Z 1043.848,A -85,B 0,C 180,E1 6064.384,E2 6064.384} C_VEL
LIN {X 0,Y 141.3,Z 1049.955,A -85,B 0,C 180,E1 6056.927,E2 6056.927} C_VEL
LIN {X 0,Y 138.254,Z 1054.134,A -85,B 0,C 180,E1 6048.991,E2 6048.991} C_VEL
LIN {X 0,Y 137.725,Z 1056.485,A -85,B 0,C 180,E1 6040.879,E2 6040.879} C_VEL
LIN {X 0,Y 138.969,Z 1057.002,A -85,B 0,C 180,E1 6033.712,E2 6033.712} C_VEL
LIN {X 0,Y 139.707,Z 1056.56,A -85,B 0,C 180,E1 6029.999,E2 6029.999} C_VEL
LIN {X 0,Y 139.005,Z 1055.038,A -85,B 0,C 180,E1 6025.461,E2 6025.461} C_VEL
LIN {X 0,Y 138.363,Z 1052.922,A -85,B 0,C 180,E1 6020.851,E2 6020.851} C_VEL
LIN {X 0,Y 138.063,Z 1052.359,A -85,B 0,C 180,E1 6013.16,E2 6013.16} C_VEL
LIN {X 0,Y 140.351,Z 1049.812,A -85,B 0,C 180,E1 6005.144,E2 6005.144} C_VEL
LIN {X 0,Y 145.232,Z 1045.552,A -85,B 0,C 180,E1 5997.864,E2 5997.864} C_VEL
LIN {X 0,Y 152.712,Z 1039.338,A -85,B 0,C 180,E1 5991.056,E2 5991.056} C_VEL
LIN {X 0,Y 162.057,Z 1031.611,A -85,B 0,C 180,E1 5985.302,E2 5985.302} C_VEL
LIN {X 0,Y 173.221,Z 1021.92,A -85,B 0,C 180,E1 5980.364,E2 5980.364} C_VEL
LIN {X 0,Y 185.15,Z 1010.815,A -85,B 0,C 180,E1 5976.423,E2 5976.423} C_VEL
LIN {X 0,Y 197.35,Z 998.172,A -85,B 0,C 180,E1 5973.282,E2 5973.282} C_VEL
LIN {X 0,Y 209.174,Z 984.467,A -85,B 0,C 180,E1 5970.904,E2 5970.904} C_VEL
LIN {X 0,Y 219.454,Z 970.766,A -85,B 0,C 180,E1 5969.214,E2 5969.214} C_VEL
LIN {X 0,Y 210.636,Z 982.072,A -85,B 0,C 180,E1 5967.109,E2 5967.109} C_VEL
LIN {X 0,Y 200.646,Z 992.75,A -85,B 0,C 180,E1 5964.431,E2 5964.431} C_VEL
LIN {X 0,Y 191.088,Z 1001.295,A -85,B 0,C 180,E1 5961.485,E2 5961.485} C_VEL
LIN {X 0,Y 180.741,Z 1008.969,A -85,B 0,C 180,E1 5957.713,E2 5957.713} C_VEL
LIN {X 0,Y 171.238,Z 1014.587,A -85,B 0,C 180,E1 5953.506,E2 5953.506} C_VEL
LIN {X 0,Y 162.229,Z 1018.604,A -85,B 0,C 180,E1 5948.506,E2 5948.506} C_VEL
LIN {X 0,Y 154.538,Z 1020.614,A -85,B 0,C 180,E1 5942.966,E2 5942.966} C_VEL
LIN {X 0,Y 148.358,Z 1020.79,A -85,B 0,C 180,E1 5936.909,E2 5936.909} C_VEL
LIN {X 0,Y 143.78,Z 1019.019,A -85,B 0,C 180,E1 5930.392,E2 5930.392} C_VEL
LIN {X 0,Y 141.026,Z 1015.596,A -85,B 0,C 180,E1 5923.947,E2 5923.947} C_VEL
LIN {X 0,Y 139.7,Z 1010.221,A -85,B 0,C 180,E1 5917.263,E2 5917.263} C_VEL
LIN {X 0,Y 139.648,Z 1003.806,A -85,B 0,C 180,E1 5911.333,E2 5911.333} C_VEL
LIN {X 0,Y 140.633,Z 995.289,A -85,B 0,C 180,E1 5905.334,E2 5905.334} C_VEL
LIN {X 0,Y 142.519,Z 985.254,A -85,B 0,C 180,E1 5899.8,E2 5899.8} C_VEL
LIN {X 0,Y 145.213,Z 973.199,A -85,B 0,C 180,E1 5894.615,E2 5894.615} C_VEL
LIN {X 0,Y 148.194,Z 960.357,A -85,B 0,C 180,E1 5890.322,E2 5890.322} C_VEL
LIN {X 0,Y 151.511,Z 945.503,A -85,B 0,C 180,E1 5886.438,E2 5886.438} C_VEL
LIN {X 0,Y 152.433,Z 942.199,A -85,B 0,C 180,E1 5885.493,E2 5885.493} C_VEL
LIN {X 0,Y 153.407,Z 941.696,A -85,B 0,C 180,E1 5884.791,E2 5884.791} C_VEL
LIN {X 0,Y 156.203,Z 941.076,A -85,B 0,C 180,E1 5883.68,E2 5883.68} C_VEL
LIN {X 0,Y 160.366,Z 938.818,A -85,B 0,C 180,E1 5882.678,E2 5882.678} C_VEL
LIN {X 0,Y 164.096,Z 937.846,A -85,B 0,C 180,E1 5881.455,E2 5881.455} C_VEL
LIN {X 0,Y 168.33,Z 935.584,A -85,B 0,C 180,E1 5880.537,E2 5880.537} C_VEL
LIN {X 0,Y 170.097,Z 934.461,A -85,B 0,C 180,E1 5880.219,E2 5880.219} C_VEL
LIN {X 0,Y 174.991,Z 932.483,A -85,B 0,C 180,E1 5879.047,E2 5879.047} C_VEL
LIN {X 0,Y 177.932,Z 930.906,A -85,B 0,C 180,E1 5878.491,E2 5878.491} C_VEL
LIN {X 0,Y 172.212,Z 946.114,A -85,B 0,C 180,E1 5875.63,E2 5875.63} C_VEL
LIN {X 0,Y 166.294,Z 959.795,A -85,B 0,C 180,E1 5872.26,E2 5872.26} C_VEL
LIN {X 0,Y 160.161,Z 972.353,A -85,B 0,C 180,E1 5868.189,E2 5868.189} C_VEL
LIN {X 0,Y 154.1,Z 983.834,A -85,B 0,C 180,E1 5863.277,E2 5863.277} C_VEL
LIN {X 0,Y 148.811,Z 993.587,A -85,B 0,C 180,E1 5857.724,E2 5857.724} C_VEL
LIN {X 0,Y 144.602,Z 1001.509,A -85,B 0,C 180,E1 5851.586,E2 5851.586} C_VEL
LIN {X 0,Y 141.647,Z 1007.887,A -85,B 0,C 180,E1 5844.736,E2 5844.736} C_VEL
LIN {X 0,Y 140.236,Z 1012.437,A -85,B 0,C 180,E1 5837.634,E2 5837.634} C_VEL
LIN {X 0,Y 140.371,Z 1015.211,A -85,B 0,C 180,E1 5830.442,E2 5830.442} C_VEL
LIN {X 0,Y 142.121,Z 1016.256,A -85,B 0,C 180,E1 5823.241,E2 5823.241} C_VEL
LIN {X 0,Y 145.878,Z 1015.506,A -85,B 0,C 180,E1 5815.805,E2 5815.805} C_VEL
LIN {X 0,Y 151.284,Z 1012.968,A -85,B 0,C 180,E1 5809.134,E2 5809.134} C_VEL
LIN {X 0,Y 157.952,Z 1008.763,A -85,B 0,C 180,E1 5803.285,E2 5803.285} C_VEL
LIN {X 0,Y 166.061,Z 1002.638,A -85,B 0,C 180,E1 5797.891,E2 5797.891} C_VEL
LIN {X 0,Y 174.722,Z 995.05,A -85,B 0,C 180,E1 5793.324,E2 5793.324} C_VEL
LIN {X 0,Y 184.112,Z 985.576,A -85,B 0,C 180,E1 5789.26,E2 5789.26} C_VEL
LIN {X 0,Y 193.357,Z 974.679,A -85,B 0,C 180,E1 5785.875,E2 5785.875} C_VEL
LIN {X 0,Y 202.144,Z 962.583,A -85,B 0,C 180,E1 5783.074,E2 5783.074} C_VEL
LIN {X 0,Y 210.543,Z 948.946,A -85,B 0,C 180,E1 5780.686,E2 5780.686} C_VEL
LIN {X 0,Y 218.135,Z 934.122,A -85,B 0,C 180,E1 5778.715,E2 5778.715} C_VEL
LIN {X 0,Y 224.469,Z 918.782,A -85,B 0,C 180,E1 5777.168,E2 5777.168} C_VEL
LIN {X 0,Y 229.762,Z 902.166,A -85,B 0,C 180,E1 5775.905,E2 5775.905} C_VEL
LIN {X 0,Y 233.815,Z 884.402,A -85,B 0,C 180,E1 5774.918,E2 5774.918} C_VEL
LIN {X 0,Y 236.324,Z 866.621,A -85,B 0,C 180,E1 5774.244,E2 5774.244} C_VEL
LIN {X 0,Y 243.315,Z 797.118,A -85,B 0,C 180,E1 5772.58,E2 5772.58} C_VEL
LIN {X 0,Y 240.376,Z 790.111,A -85,B 0,C 180,E1 5769.518,E2 5769.518} C_VEL
LIN {X 0,Y 237.884,Z 784.391,A -85,B 0,C 180,E1 5766.153,E2 5766.153} C_VEL
LIN {X 0,Y 236.175,Z 781.055,A -85,B 0,C 180,E1 5763.155,E2 5763.155} C_VEL
LIN {X 0,Y 235.393,Z 779.169,A -85,B 0,C 180,E1 5761.217,E2 5761.217} C_VEL
LIN {X 0,Y 234.459,Z 777.044,A -85,B 0,C 180,E1 5756.281,E2 5756.281} C_VEL
LIN {X 0,Y 234.695,Z 777.505,A -85,B 0,C 180,E1 5752.411,E2 5752.411} C_VEL
LIN {X 0,Y 236.343,Z 780.698,A -85,B 0,C 180,E1 5747.54,E2 5747.54} C_VEL
LIN {X 0,Y 238.989,Z 786.127,A -85,B 0,C 180,E1 5743.222,E2 5743.222} C_VEL
LIN {X 0,Y 241.701,Z 792.141,A -85,B 0,C 180,E1 5740.045,E2 5740.045} C_VEL
LIN {X 0,Y 243.701,Z 796.963,A -85,B 0,C 180,E1 5738.064,E2 5738.064} C_VEL
LIN {X 0,Y 241.654,Z 817.078,A -85,B 0,C 180,E1 5737.614,E2 5737.614} C_VEL
LIN {X 0,Y 240.551,Z 824.766,A -85,B 0,C 180,E1 5737.671,E2 5737.671} C_VEL
LIN {X 0,Y 236.507,Z 845.236,A -85,B 0,C 180,E1 5738.642,E2 5738.642} C_VEL
LIN {X 0,Y 235.615,Z 851.83,A -85,B 0,C 180,E1 5738.656,E2 5738.656} C_VEL
LIN {X 0,Y 231.318,Z 890.972,A -85,B 0,C 180,E1 5737.728,E2 5737.728} C_VEL
LIN {X 0,Y 227.498,Z 909.745,A -85,B 0,C 180,E1 5737.096,E2 5737.096} C_VEL
LIN {X 0,Y 222.234,Z 927.388,A -85,B 0,C 180,E1 5736.286,E2 5736.286} C_VEL
LIN {X 0,Y 215.784,Z 943.873,A -85,B 0,C 180,E1 5735.255,E2 5735.255} C_VEL
LIN {X 0,Y 207.775,Z 960.443,A -85,B 0,C 180,E1 5733.827,E2 5733.827} C_VEL
LIN {X 0,Y 198.77,Z 975.914,A -85,B 0,C 180,E1 5731.981,E2 5731.981} C_VEL
LIN {X 0,Y 188.92,Z 990.356,A -85,B 0,C 180,E1 5729.617,E2 5729.617} C_VEL
LIN {X 0,Y 178.434,Z 1003.765,A -85,B 0,C 180,E1 5726.607,E2 5726.607} C_VEL
LIN {X 0,Y 167.954,Z 1015.696,A -85,B 0,C 180,E1 5722.912,E2 5722.912} C_VEL
LIN {X 0,Y 157.785,Z 1026.218,A -85,B 0,C 180,E1 5718.394,E2 5718.394} C_VEL
LIN {X 0,Y 148.36,Z 1035.31,A -85,B 0,C 180,E1 5712.895,E2 5712.895} C_VEL
LIN {X 0,Y 140.227,Z 1042.924,A -85,B 0,C 180,E1 5706.285,E2 5706.285} C_VEL
LIN {X 0,Y 134.012,Z 1048.906,A -85,B 0,C 180,E1 5698.521,E2 5698.521} C_VEL
LIN {X 0,Y 130.528,Z 1053.002,A -85,B 0,C 180,E1 5690.163,E2 5690.163} C_VEL
LIN {X 0,Y 129.748,Z 1055.276,A -85,B 0,C 180,E1 5681.557,E2 5681.557} C_VEL
LIN {X 0,Y 130.98,Z 1055.727,A -85,B 0,C 180,E1 5673.938,E2 5673.938} C_VEL
LIN {X 0,Y 131.809,Z 1055.259,A -85,B 0,C 180,E1 5669.999,E2 5669.999} C_VEL
LIN {X 0,Y 131.013,Z 1053.674,A -85,B 0,C 180,E1 5665.183,E2 5665.183} C_VEL
LIN {X 0,Y 130.36,Z 1051.271,A -85,B 0,C 180,E1 5659.838,E2 5659.838} C_VEL
LIN {X 0,Y 130.345,Z 1050.901,A -85,B 0,C 180,E1 5651.668,E2 5651.668} C_VEL
LIN {X 0,Y 133.171,Z 1048.561,A -85,B 0,C 180,E1 5643.224,E2 5643.224} C_VEL
LIN {X 0,Y 138.991,Z 1044.419,A -85,B 0,C 180,E1 5635.367,E2 5635.367} C_VEL
LIN {X 0,Y 147.46,Z 1038.427,A -85,B 0,C 180,E1 5628.355,E2 5628.355} C_VEL
LIN {X 0,Y 158.259,Z 1030.546,A -85,B 0,C 180,E1 5622.336,E2 5622.336} C_VEL
LIN {X 0,Y 169.578,Z 1021.804,A -85,B 0,C 180,E1 5617.805,E2 5617.805} C_VEL
LIN {X 0,Y 182.147,Z 1011.154,A -85,B 0,C 180,E1 5614.014,E2 5614.014} C_VEL
LIN {X 0,Y 194.892,Z 999.179,A -85,B 0,C 180,E1 5611.043,E2 5611.043} C_VEL
LIN {X 0,Y 207.137,Z 986.127,A -85,B 0,C 180,E1 5608.791,E2 5608.791} C_VEL
LIN {X 0,Y 196.867,Z 996.132,A -85,B 0,C 180,E1 5606.222,E2 5606.222} C_VEL
LIN {X 0,Y 185.345,Z 1005.402,A -85,B 0,C 180,E1 5602.855,E2 5602.855} C_VEL
LIN {X 0,Y 174.528,Z 1012.376,A -85,B 0,C 180,E1 5599.059,E2 5599.059} C_VEL
LIN {X 0,Y 164.322,Z 1017.56,A -85,B 0,C 180,E1 5594.649,E2 5594.649} C_VEL
LIN {X 0,Y 154.59,Z 1021.011,A -85,B 0,C 180,E1 5589.305,E2 5589.305} C_VEL
LIN {X 0,Y 147.068,Z 1022.379,A -85,B 0,C 180,E1 5583.898,E2 5583.898} C_VEL
LIN {X 0,Y 140.572,Z 1022.029,A -85,B 0,C 180,E1 5577.553,E2 5577.553} C_VEL
LIN {X 0,Y 136.041,Z 1020.005,A -85,B 0,C 180,E1 5571.12,E2 5571.12} C_VEL
LIN {X 0,Y 132.958,Z 1015.883,A -85,B 0,C 180,E1 5563.844,E2 5563.844} C_VEL
LIN {X 0,Y 131.7,Z 1010.504,A -85,B 0,C 180,E1 5557.219,E2 5557.219} C_VEL
LIN {X 0,Y 131.723,Z 1003.088,A -85,B 0,C 180,E1 5550.435,E2 5550.435} C_VEL
LIN {X 0,Y 132.837,Z 994.544,A -85,B 0,C 180,E1 5544.383,E2 5544.383} C_VEL
LIN {X 0,Y 134.995,Z 983.74,A -85,B 0,C 180,E1 5538.425,E2 5538.425} C_VEL
LIN {X 0,Y 137.697,Z 972.143,A -85,B 0,C 180,E1 5533.436,E2 5533.436} C_VEL
LIN {X 0,Y 140.861,Z 959.016,A -85,B 0,C 180,E1 5528.989,E2 5528.989} C_VEL
LIN {X 0,Y 142.906,Z 950.962,A -85,B 0,C 180,E1 5526.575,E2 5526.575} C_VEL
LIN {X 0,Y 144.022,Z 950.408,A -85,B 0,C 180,E1 5525.675,E2 5525.675} C_VEL
LIN {X 0,Y 146.751,Z 949.858,A -85,B 0,C 180,E1 5524.47,E2 5524.47} C_VEL
LIN {X 0,Y 150.108,Z 948.227,A -85,B 0,C 180,E1 5523.564,E2 5523.564} C_VEL
LIN {X 0,Y 153.606,Z 947.599,A -85,B 0,C 180,E1 5522.198,E2 5522.198} C_VEL
LIN {X 0,Y 158.592,Z 945.303,A -85,B 0,C 180,E1 5520.97,E2 5520.97} C_VEL
LIN {X 0,Y 164.156,Z 943.511,A -85,B 0,C 180,E1 5519.423,E2 5519.423} C_VEL
LIN {X 0,Y 168.536,Z 941.189,A -85,B 0,C 180,E1 5518.593,E2 5518.593} C_VEL
LIN {X 0,Y 162.373,Z 955.574,A -85,B 0,C 180,E1 5515.34,E2 5515.34} C_VEL
LIN {X 0,Y 155.935,Z 968.636,A -85,B 0,C 180,E1 5511.439,E2 5511.439} C_VEL
LIN {X 0,Y 149.463,Z 980.601,A -85,B 0,C 180,E1 5506.719,E2 5506.719} C_VEL
LIN {X 0,Y 143.544,Z 990.993,A -85,B 0,C 180,E1 5501.248,E2 5501.248} C_VEL
LIN {X 0,Y 138.784,Z 999.253,A -85,B 0,C 180,E1 5495.375,E2 5495.375} C_VEL
LIN {X 0,Y 135.027,Z 1006.302,A -85,B 0,C 180,E1 5488.545,E2 5488.545} C_VEL
LIN {X 0,Y 132.817,Z 1011.581,A -85,B 0,C 180,E1 5481.342,E2 5481.342} C_VEL
LIN {X 0,Y 132.192,Z 1015.245,A -85,B 0,C 180,E1 5473.75,E2 5473.75} C_VEL
LIN {X 0,Y 133.255,Z 1017.152,A -85,B 0,C 180,E1 5466.099,E2 5466.099} C_VEL
LIN {X 0,Y 136.265,Z 1017.338,A -85,B 0,C 180,E1 5458.34,E2 5458.34} C_VEL
LIN {X 0,Y 141.274,Z 1015.697,A -85,B 0,C 180,E1 5450.959,E2 5450.959} C_VEL
LIN {X 0,Y 147.59,Z 1012.474,A -85,B 0,C 180,E1 5444.658,E2 5444.658} C_VEL
LIN {X 0,Y 155.419,Z 1007.441,A -85,B 0,C 180,E1 5438.884,E2 5438.884} C_VEL
LIN {X 0,Y 164.582,Z 1000.445,A -85,B 0,C 180,E1 5433.667,E2 5433.667} C_VEL
LIN {X 0,Y 174.216,Z 991.868,A -85,B 0,C 180,E1 5429.268,E2 5429.268} C_VEL
LIN {X 0,Y 183.989,Z 981.757,A -85,B 0,C 180,E1 5425.566,E2 5425.566} C_VEL
LIN {X 0,Y 193.629,Z 969.989,A -85,B 0,C 180,E1 5422.436,E2 5422.436} C_VEL
LIN {X 0,Y 202.423,Z 957.379,A -85,B 0,C 180,E1 5419.928,E2 5419.928} C_VEL
LIN {X 0,Y 210.577,Z 943.474,A -85,B 0,C 180,E1 5417.824,E2 5417.824} C_VEL
LIN {X 0,Y 217.978,Z 928.129,A -85,B 0,C 180,E1 5416.062,E2 5416.062} C_VEL
LIN {X 0,Y 223.861,Z 912.786,A -85,B 0,C 180,E1 5414.723,E2 5414.723} C_VEL
LIN {X 0,Y 228.781,Z 895.704,A -85,B 0,C 180,E1 5413.607,E2 5413.607} C_VEL
LIN {X 0,Y 232.304,Z 877.795,A -85,B 0,C 180,E1 5412.768,E2 5412.768} C_VEL
LIN {X 0,Y 235.138,Z 852.465,A -85,B 0,C 180,E1 5412.018,E2 5412.018} C_VEL
LIN {X 0,Y 240.415,Z 801.722,A -85,B 0,C 180,E1 5410.847,E2 5410.847} C_VEL
LIN {X 0,Y 237.789,Z 795.077,A -85,B 0,C 180,E1 5407.612,E2 5407.612} C_VEL
LIN {X 0,Y 235.762,Z 790.404,A -85,B 0,C 180,E1 5404.379,E2 5404.379} C_VEL
LIN {X 0,Y 234.195,Z 786.899,A -85,B 0,C 180,E1 5400.734,E2 5400.734} C_VEL
LIN {X 0,Y 233.441,Z 784.97,A -85,B 0,C 180,E1 5396.071,E2 5396.071} C_VEL
LIN {X 0,Y 233.684,Z 785.515,A -85,B 0,C 180,E1 5392.378,E2 5392.378} C_VEL
LIN {X 0,Y 235.15,Z 788.563,A -85,B 0,C 180,E1 5387.85,E2 5387.85} C_VEL
LIN {X 0,Y 237.441,Z 793.516,A -85,B 0,C 180,E1 5383.864,E2 5383.864} C_VEL
LIN {X 0,Y 239.87,Z 799.308,A -85,B 0,C 180,E1 5380.774,E2 5380.774} C_VEL
LIN {X 0,Y 240.785,Z 801.712,A -85,B 0,C 180,E1 5379.766,E2 5379.766} C_VEL
LIN {X 0,Y 235.615,Z 851.83,A -85,B 0,C 180,E1 5378.656,E2 5378.656} C_VEL
LIN {X 0,Y 234.547,Z 859.515,A -85,B 0,C 180,E1 5378.704,E2 5378.704} C_VEL
LIN {X 0,Y 230.537,Z 879.974,A -85,B 0,C 180,E1 5379.724,E2 5379.724} C_VEL
LIN {X 0,Y 229.496,Z 886.558,A -85,B 0,C 180,E1 5379.743,E2 5379.743} C_VEL
LIN {X 0,Y 225.976,Z 905.24,A -85,B 0,C 180,E1 5379.178,E2 5379.178} C_VEL
LIN {X 0,Y 220.911,Z 922.929,A -85,B 0,C 180,E1 5378.45,E2 5378.45} C_VEL
LIN {X 0,Y 214.306,Z 940.169,A -85,B 0,C 180,E1 5377.484,E2 5377.484} C_VEL
LIN {X 0,Y 206.186,Z 957.03,A -85,B 0,C 180,E1 5376.171,E2 5376.171} C_VEL
LIN {X 0,Y 197.189,Z 972.491,A -85,B 0,C 180,E1 5374.495,E2 5374.495} C_VEL
LIN {X 0,Y 187.127,Z 987.185,A -85,B 0,C 180,E1 5372.299,E2 5372.299} C_VEL
LIN {X 0,Y 176.376,Z 1000.695,A -85,B 0,C 180,E1 5369.504,E2 5369.504} C_VEL
LIN {X 0,Y 165.283,Z 1012.919,A -85,B 0,C 180,E1 5365.971,E2 5365.971} C_VEL
LIN {X 0,Y 154.188,Z 1023.866,A -85,B 0,C 180,E1 5361.5,E2 5361.5} C_VEL
LIN {X 0,Y 143.548,Z 1033.491,A -85,B 0,C 180,E1 5355.841,E2 5355.841} C_VEL
LIN {X 0,Y 134.549,Z 1041.227,A -85,B 0,C 180,E1 5349.171,E2 5349.171} C_VEL
LIN {X 0,Y 127.433,Z 1047.357,A -85,B 0,C 180,E1 5341.186,E2 5341.186} C_VEL
LIN {X 0,Y 123.134,Z 1051.548,A -85,B 0,C 180,E1 5332.434,E2 5332.434} C_VEL
LIN {X 0,Y 121.763,Z 1053.923,A -85,B 0,C 180,E1 5323.291,E2 5323.291} C_VEL
LIN {X 0,Y 122.872,Z 1054.471,A -85,B 0,C 180,E1 5314.666,E2 5314.666} C_VEL
LIN {X 0,Y 123.907,Z 1053.955,A -85,B 0,C 180,E1 5309.999,E2 5309.999} C_VEL
LIN {X 0,Y 122.934,Z 1052.123,A -85,B 0,C 180,E1 5304.398,E2 5304.398} C_VEL
LIN {X 0,Y 122.391,Z 1049.548,A -85,B 0,C 180,E1 5298.611,E2 5298.611} C_VEL
LIN {X 0,Y 122.854,Z 1049.275,A -85,B 0,C 180,E1 5289.378,E2 5289.378} C_VEL
LIN {X 0,Y 126.438,Z 1047.151,A -85,B 0,C 180,E1 5280.639,E2 5280.639} C_VEL
LIN {X 0,Y 133.591,Z 1042.951,A -85,B 0,C 180,E1 5272.139,E2 5272.139} C_VEL
LIN {X 0,Y 143.138,Z 1037.203,A -85,B 0,C 180,E1 5265.128,E2 5265.128} C_VEL
LIN {X 0,Y 154.942,Z 1029.578,A -85,B 0,C 180,E1 5259.25,E2 5259.25} C_VEL
LIN {X 0,Y 167.799,Z 1020.604,A -85,B 0,C 180,E1 5254.683,E2 5254.683} C_VEL
LIN {X 0,Y 181.108,Z 1010.279,A -85,B 0,C 180,E1 5251.158,E2 5251.158} C_VEL
LIN {X 0,Y 194.569,Z 998.497,A -85,B 0,C 180,E1 5248.393,E2 5248.393} C_VEL
LIN {X 0,Y 182.8,Z 1007.314,A -85,B 0,C 180,E1 5245.254,E2 5245.254} C_VEL
LIN {X 0,Y 170.58,Z 1014.578,A -85,B 0,C 180,E1 5241.309,E2 5241.309} C_VEL
LIN {X 0,Y 159.999,Z 1019.406,A -85,B 0,C 180,E1 5237.08,E2 5237.08} C_VEL
LIN {X 0,Y 149.258,Z 1022.788,A -85,B 0,C 180,E1 5231.593,E2 5231.593} C_VEL
LIN {X 0,Y 140.583,Z 1023.982,A -85,B 0,C 180,E1 5225.714,E2 5225.714} C_VEL
LIN {X 0,Y 133.549,Z 1023.392,A -85,B 0,C 180,E1 5219.141,E2 5219.141} C_VEL
LIN {X 0,Y 128.274,Z 1020.833,A -85,B 0,C 180,E1 5211.87,E2 5211.87} C_VEL
LIN {X 0,Y 125.168,Z 1016.748,A -85,B 0,C 180,E1 5204.715,E2 5204.715} C_VEL
LIN {X 0,Y 123.694,Z 1010.634,A -85,B 0,C 180,E1 5197.169,E2 5197.169} C_VEL
LIN {X 0,Y 123.715,Z 1003.507,A -85,B 0,C 180,E1 5190.461,E2 5190.461} C_VEL
LIN {X 0,Y 124.966,Z 994.179,A -85,B 0,C 180,E1 5183.694,E2 5183.694} C_VEL
LIN {X 0,Y 127.195,Z 983.495,A -85,B 0,C 180,E1 5177.641,E2 5177.641} C_VEL
LIN {X 0,Y 130.368,Z 970.49,A -85,B 0,C 180,E1 5171.93,E2 5171.93} C_VEL
LIN {X 0,Y 133.399,Z 958.881,A -85,B 0,C 180,E1 5167.778,E2 5167.778} C_VEL
LIN {X 0,Y 134.092,Z 958.382,A -85,B 0,C 180,E1 5167.073,E2 5167.073} C_VEL
LIN {X 0,Y 136.597,Z 958.078,A -85,B 0,C 180,E1 5165.658,E2 5165.658} C_VEL
LIN {X 0,Y 140.093,Z 956.714,A -85,B 0,C 180,E1 5164.477,E2 5164.477} C_VEL
LIN {X 0,Y 143.936,Z 956.085,A -85,B 0,C 180,E1 5162.802,E2 5162.802} C_VEL
LIN {X 0,Y 148.715,Z 954.35,A -85,B 0,C 180,E1 5161.364,E2 5161.364} C_VEL
LIN {X 0,Y 153.396,Z 953.037,A -85,B 0,C 180,E1 5159.896,E2 5159.896} C_VEL
LIN {X 0,Y 158.459,Z 951.001,A -85,B 0,C 180,E1 5158.707,E2 5158.707} C_VEL
LIN {X 0,Y 158.918,Z 950.903,A -85,B 0,C 180,E1 5158.567,E2 5158.567} C_VEL
LIN {X 0,Y 152.208,Z 964.528,A -85,B 0,C 180,E1 5154.862,E2 5154.862} C_VEL
LIN {X 0,Y 145.556,Z 976.641,A -85,B 0,C 180,E1 5150.509,E2 5150.509} C_VEL
LIN {X 0,Y 139.227,Z 987.34,A -85,B 0,C 180,E1 5145.411,E2 5145.411} C_VEL
LIN {X 0,Y 133.559,Z 996.577,A -85,B 0,C 180,E1 5139.481,E2 5139.481} C_VEL
LIN {X 0,Y 128.933,Z 1004.343,A -85,B 0,C 180,E1 5132.668,E2 5132.668} C_VEL
LIN {X 0,Y 125.734,Z 1010.615,A -85,B 0,C 180,E1 5124.983,E2 5124.983} C_VEL
LIN {X 0,Y 124.324,Z 1015.057,A -85,B 0,C 180,E1 5116.987,E2 5116.987} C_VEL
LIN {X 0,Y 124.724,Z 1017.712,A -85,B 0,C 180,E1 5108.855,E2 5108.855} C_VEL
LIN {X 0,Y 127.041,Z 1018.688,A -85,B 0,C 180,E1 5100.795,E2 5100.795} C_VEL
LIN {X 0,Y 131.37,Z 1017.956,A -85,B 0,C 180,E1 5093.041,E2 5093.041} C_VEL
LIN {X 0,Y 137.702,Z 1015.452,A -85,B 0,C 180,E1 5085.81,E2 5085.81} C_VEL
LIN {X 0,Y 145.349,Z 1011.315,A -85,B 0,C 180,E1 5079.607,E2 5079.607} C_VEL
LIN {X 0,Y 154.428,Z 1005.297,A -85,B 0,C 180,E1 5074.031,E2 5074.031} C_VEL
LIN {X 0,Y 164.735,Z 997.216,A -85,B 0,C 180,E1 5069.074,E2 5069.074} C_VEL
LIN {X 0,Y 174.598,Z 988.157,A -85,B 0,C 180,E1 5065.204,E2 5065.204} C_VEL
LIN {X 0,Y 184.738,Z 977.244,A -85,B 0,C 180,E1 5061.844,E2 5061.844} C_VEL
LIN {X 0,Y 194.156,Z 965.287,A -85,B 0,C 180,E1 5059.135,E2 5059.135} C_VEL
LIN {X 0,Y 203.128,Z 951.799,A -85,B 0,C 180,E1 5056.837,E2 5056.837} C_VEL
LIN {X 0,Y 211.132,Z 937.304,A -85,B 0,C 180,E1 5054.967,E2 5054.967} C_VEL
LIN {X 0,Y 217.964,Z 922.073,A -85,B 0,C 180,E1 5053.471,E2 5053.471} C_VEL
LIN {X 0,Y 223.579,Z 906.053,A -85,B 0,C 180,E1 5052.275,E2 5052.275} C_VEL
LIN {X 0,Y 227.986,Z 888.666,A -85,B 0,C 180,E1 5051.316,E2 5051.316} C_VEL
LIN {X 0,Y 230.96,Z 870.217,A -85,B 0,C 180,E1 5050.609,E2 5050.609} C_VEL
LIN {X 0,Y 237.793,Z 806.693,A -85,B 0,C 180,E1 5049.134,E2 5049.134} C_VEL
LIN {X 0,Y 235.67,Z 801.12,A -85,B 0,C 180,E1 5046.089,E2 5046.089} C_VEL
LIN {X 0,Y 234.402,Z 797.954,A -85,B 0,C 180,E1 5043.791,E2 5043.791} C_VEL
LIN {X 0,Y 233.103,Z 794.762,A -85,B 0,C 180,E1 5040.492,E2 5040.492} C_VEL
LIN {X 0,Y 232.434,Z 792.906,A -85,B 0,C 180,E1 5036.054,E2 5036.054} C_VEL
LIN {X 0,Y 232.637,Z 793.4,A -85,B 0,C 180,E1 5032.592,E2 5032.592} C_VEL
LIN {X 0,Y 233.916,Z 796.275,A -85,B 0,C 180,E1 5028.286,E2 5028.286} C_VEL
LIN {X 0,Y 235.96,Z 801.013,A -85,B 0,C 180,E1 5024.454,E2 5024.454} C_VEL
LIN {X 0,Y 238.079,Z 806.476,A -85,B 0,C 180,E1 5021.514,E2 5021.514} C_VEL
LIN {X 0,Y 229.496,Z 886.558,A -85,B 0,C 180,E1 5019.743,E2 5019.743} C_VEL
LIN {X 0,Y 228.049,Z 894.193,A -85,B 0,C 180,E1 5019.781,E2 5019.781} C_VEL
LIN {X 0,Y 222.979,Z 909.948,A -85,B 0,C 180,E1 5020.508,E2 5020.508} C_VEL
LIN {X 0,Y 219.945,Z 918.306,A -85,B 0,C 180,E1 5020.613,E2 5020.613} C_VEL
LIN {X 0,Y 219.224,Z 920.392,A -85,B 0,C 180,E1 5020.546,E2 5020.546} C_VEL
LIN {X 0,Y 212.718,Z 937.469,A -85,B 0,C 180,E1 5019.672,E2 5019.672} C_VEL
LIN {X 0,Y 204.76,Z 953.984,A -85,B 0,C 180,E1 5018.507,E2 5018.507} C_VEL
LIN {X 0,Y 195.574,Z 969.68,A -85,B 0,C 180,E1 5016.96,E2 5016.96} C_VEL
LIN {X 0,Y 185.413,Z 984.328,A -85,B 0,C 180,E1 5014.951,E2 5014.951} C_VEL
LIN {X 0,Y 174.784,Z 997.503,A -85,B 0,C 180,E1 5012.458,E2 5012.458} C_VEL
LIN {X 0,Y 163.87,Z 1009.348,A -85,B 0,C 180,E1 5009.35,E2 5009.35} C_VEL
LIN {X 0,Y 152.205,Z 1020.57,A -85,B 0,C 180,E1 5005.198,E2 5005.198} C_VEL
LIN {X 0,Y 140.978,Z 1030.218,A -85,B 0,C 180,E1 4999.992,E2 4999.992} C_VEL
LIN {X 0,Y 130.753,Z 1038.344,A -85,B 0,C 180,E1 4993.488,E2 4993.488} C_VEL
LIN {X 0,Y 122.256,Z 1044.897,A -85,B 0,C 180,E1 4985.496,E2 4985.496} C_VEL
LIN {X 0,Y 116.563,Z 1049.52,A -85,B 0,C 180,E1 4976.489,E2 4976.489} C_VEL
LIN {X 0,Y 114.001,Z 1052.315,A -85,B 0,C 180,E1 4966.823,E2 4966.823} C_VEL
LIN {X 0,Y 114.45,Z 1053.271,A -85,B 0,C 180,E1 4957.024,E2 4957.024} C_VEL
LIN {X 0,Y 115.983,Z 1052.678,A -85,B 0,C 180,E1 4950.196,E2 4950.196} C_VEL
LIN {X 0,Y 115.007,Z 1050.918,A -85,B 0,C 180,E1 4944.511,E2 4944.511} C_VEL
LIN {X 0,Y 114.491,Z 1047.771,A -85,B 0,C 180,E1 4937.388,E2 4937.388} C_VEL
LIN {X 0,Y 115.361,Z 1047.712,A -85,B 0,C 180,E1 4927.581,E2 4927.581} C_VEL
LIN {X 0,Y 119.997,Z 1045.702,A -85,B 0,C 180,E1 4917.772,E2 4917.772} C_VEL
LIN {X 0,Y 127.833,Z 1041.951,A -85,B 0,C 180,E1 4909.348,E2 4909.348} C_VEL
LIN {X 0,Y 138.705,Z 1036.314,A -85,B 0,C 180,E1 4902.055,E2 4902.055} C_VEL
LIN {X 0,Y 151.403,Z 1029.152,A -85,B 0,C 180,E1 4896.322,E2 4896.322} C_VEL
LIN {X 0,Y 164.983,Z 1020.586,A -85,B 0,C 180,E1 4891.955,E2 4891.955} C_VEL
LIN {X 0,Y 179.713,Z 1010.17,A -85,B 0,C 180,E1 4888.469,E2 4888.469} C_VEL
LIN {X 0,Y 181.852,Z 1008.552,A -85,B 0,C 180,E1 4888.024,E2 4888.024} C_VEL
LIN {X 0,Y 169.274,Z 1015.667,A -85,B 0,C 180,E1 4884.423,E2 4884.423} C_VEL
LIN {X 0,Y 157.144,Z 1020.911,A -85,B 0,C 180,E1 4880.095,E2 4880.095} C_VEL
LIN {X 0,Y 145.469,Z 1024.3,A -85,B 0,C 180,E1 4874.732,E2 4874.732} C_VEL
LIN {X 0,Y 135.875,Z 1025.541,A -85,B 0,C 180,E1 4868.889,E2 4868.889} C_VEL
LIN {X 0,Y 127.921,Z 1024.991,A -85,B 0,C 180,E1 4862.239,E2 4862.239} C_VEL
LIN {X 0,Y 121.815,Z 1022.556,A -85,B 0,C 180,E1 4854.819,E2 4854.819} C_VEL
LIN {X 0,Y 117.762,Z 1018.22,A -85,B 0,C 180,E1 4846.746,E2 4846.746} C_VEL
LIN {X 0,Y 115.858,Z 1012.131,A -85,B 0,C 180,E1 4838.747,E2 4838.747} C_VEL
LIN {X 0,Y 115.625,Z 1005.079,A -85,B 0,C 180,E1 4831.6,E2 4831.6} C_VEL
LIN {X 0,Y 116.726,Z 995.846,A -85,B 0,C 180,E1 4824.374,E2 4824.374} C_VEL
LIN {X 0,Y 118.975,Z 985.041,A -85,B 0,C 180,E1 4817.753,E2 4817.753} C_VEL
LIN {X 0,Y 122.106,Z 972.468,A -85,B 0,C 180,E1 4811.826,E2 4811.826} C_VEL
LIN {X 0,Y 123.866,Z 966.184,A -85,B 0,C 180,E1 4809.2,E2 4809.2} C_VEL
LIN {X 0,Y 124.742,Z 965.751,A -85,B 0,C 180,E1 4808.23,E2 4808.23} C_VEL
LIN {X 0,Y 127.585,Z 965.294,A -85,B 0,C 180,E1 4806.557,E2 4806.557} C_VEL
LIN {X 0,Y 130.182,Z 964.446,A -85,B 0,C 180,E1 4805.497,E2 4805.497} C_VEL
LIN {X 0,Y 134.287,Z 963.8,A -85,B 0,C 180,E1 4803.495,E2 4803.495} C_VEL
LIN {X 0,Y 137.426,Z 962.728,A -85,B 0,C 180,E1 4802.436,E2 4802.436} C_VEL
LIN {X 0,Y 142.684,Z 961.564,A -85,B 0,C 180,E1 4800.465,E2 4800.465} C_VEL
LIN {X 0,Y 146.778,Z 960.202,A -85,B 0,C 180,E1 4799.313,E2 4799.313} C_VEL
LIN {X 0,Y 149.159,Z 959.723,A -85,B 0,C 180,E1 4798.52,E2 4798.52} C_VEL
LIN {X 0,Y 142.28,Z 972.192,A -85,B 0,C 180,E1 4794.496,E2 4794.496} C_VEL
LIN {X 0,Y 135.165,Z 983.925,A -85,B 0,C 180,E1 4789.445,E2 4789.445} C_VEL
LIN {X 0,Y 128.616,Z 994.043,A -85,B 0,C 180,E1 4783.488,E2 4783.488} C_VEL
LIN {X 0,Y 123.05,Z 1002.628,A -85,B 0,C 180,E1 4776.533,E2 4776.533} C_VEL
LIN {X 0,Y 119.012,Z 1009.493,A -85,B 0,C 180,E1 4768.781,E2 4768.781} C_VEL
LIN {X 0,Y 116.792,Z 1014.528,A -85,B 0,C 180,E1 4760.64,E2 4760.64} C_VEL
LIN {X 0,Y 116.42,Z 1017.937,A -85,B 0,C 180,E1 4751.991,E2 4751.991} C_VEL
LIN {X 0,Y 118.08,Z 1019.669,A -85,B 0,C 180,E1 4743.336,E2 4743.336} C_VEL
LIN {X 0,Y 121.888,Z 1019.719,A -85,B 0,C 180,E1 4734.957,E2 4734.957} C_VEL
LIN {X 0,Y 127.841,Z 1018.037,A -85,B 0,C 180,E1 4727.124,E2 4727.124} C_VEL
LIN {X 0,Y 135.788,Z 1014.466,A -85,B 0,C 180,E1 4720.024,E2 4720.024} C_VEL
LIN {X 0,Y 145.141,Z 1009.085,A -85,B 0,C 180,E1 4713.919,E2 4713.919} C_VEL
LIN {X 0,Y 155.232,Z 1002.116,A -85,B 0,C 180,E1 4708.84,E2 4708.84} C_VEL
LIN {X 0,Y 165.935,Z 993.382,A -85,B 0,C 180,E1 4704.515,E2 4704.515} C_VEL
LIN {X 0,Y 176.631,Z 983.022,A -85,B 0,C 180,E1 4700.932,E2 4700.932} C_VEL
LIN {X 0,Y 186.385,Z 971.918,A -85,B 0,C 180,E1 4698.129,E2 4698.129} C_VEL
LIN {X 0,Y 196.236,Z 958.65,A -85,B 0,C 180,E1 4695.639,E2 4695.639} C_VEL
LIN {X 0,Y 204.788,Z 944.838,A -85,B 0,C 180,E1 4693.69,E2 4693.69} C_VEL
LIN {X 0,Y 212.645,Z 929.386,A -85,B 0,C 180,E1 4692.039,E2 4692.039} C_VEL
LIN {X 0,Y 219.057,Z 913.313,A -85,B 0,C 180,E1 4690.743,E2 4690.743} C_VEL
LIN {X 0,Y 224.207,Z 896.108,A -85,B 0,C 180,E1 4689.706,E2 4689.706} C_VEL
LIN {X 0,Y 227.853,Z 878.213,A -85,B 0,C 180,E1 4688.931,E2 4688.931} C_VEL
LIN {X 0,Y 231.381,Z 847.784,A -85,B 0,C 180,E1 4688.113,E2 4688.113} C_VEL
LIN {X 0,Y 235.357,Z 811.743,A -85,B 0,C 180,E1 4687.323,E2 4687.323} C_VEL
LIN {X 0,Y 233.371,Z 806.077,A -85,B 0,C 180,E1 4683.808,E2 4683.808} C_VEL
LIN {X 0,Y 231.949,Z 802.503,A -85,B 0,C 180,E1 4680,E2 4680} C_VEL
LIN {X 0,Y 231.427,Z 800.842,A -85,B 0,C 180,E1 4676.037,E2 4676.037} C_VEL
LIN {X 0,Y 231.594,Z 801.285,A -85,B 0,C 180,E1 4672.808,E2 4672.808} C_VEL
LIN {X 0,Y 232.696,Z 803.986,A -85,B 0,C 180,E1 4668.726,E2 4668.726} C_VEL
LIN {X 0,Y 234.505,Z 808.508,A -85,B 0,C 180,E1 4665.052,E2 4665.052} C_VEL
LIN {X 0,Y 235.596,Z 811.792,A -85,B 0,C 180,E1 4663.28,E2 4663.28} C_VEL
LIN {X 0,Y 226.977,Z 888.455,A -85,B 0,C 180,E1 4661.626,E2 4661.626} C_VEL
LIN {X 0,Y 223.133,Z 906.953,A -85,B 0,C 180,E1 4661.067,E2 4661.067} C_VEL
LIN {X 0,Y 219.224,Z 920.392,A -85,B 0,C 180,E1 4660.546,E2 4660.546} C_VEL
LIN {X 0,Y 216.357,Z 927.664,A -85,B 0,C 180,E1 4660.463,E2 4660.463} C_VEL
LIN {X 0,Y 207.485,Z 944.313,A -85,B 0,C 180,E1 4660.995,E2 4660.995} C_VEL
LIN {X 0,Y 203.646,Z 951.037,A -85,B 0,C 180,E1 4660.852,E2 4660.852} C_VEL
LIN {X 0,Y 203.118,Z 951.974,A -85,B 0,C 180,E1 4660.786,E2 4660.786} C_VEL
LIN {X 0,Y 193.848,Z 967.609,A -85,B 0,C 180,E1 4659.374,E2 4659.374} C_VEL
LIN {X 0,Y 183,Z 982.928,A -85,B 0,C 180,E1 4657.422,E2 4657.422} C_VEL
LIN {X 0,Y 172.015,Z 996.151,A -85,B 0,C 180,E1 4655.061,E2 4655.061} C_VEL
LIN {X 0,Y 160.663,Z 1008.027,A -85,B 0,C 180,E1 4652.092,E2 4652.092} C_VEL
LIN {X 0,Y 148.427,Z 1019.275,A -85,B 0,C 180,E1 4648.078,E2 4648.078} C_VEL
LIN {X 0,Y 136.508,Z 1028.935,A -85,B 0,C 180,E1 4642.974,E2 4642.974} C_VEL
LIN {X 0,Y 125.471,Z 1037.064,A -85,B 0,C 180,E1 4636.481,E2 4636.481} C_VEL
LIN {X 0,Y 116.074,Z 1043.602,A -85,B 0,C 180,E1 4628.33,E2 4628.33} C_VEL
LIN {X 0,Y 109.524,Z 1048.226,A -85,B 0,C 180,E1 4618.935,E2 4618.935} C_VEL
LIN {X 0,Y 106.274,Z 1051.028,A -85,B 0,C 180,E1 4608.654,E2 4608.654} C_VEL
LIN {X 0,Y 106.345,Z 1051.997,A -85,B 0,C 180,E1 4598.106,E2 4598.106} C_VEL
LIN {X 0,Y 108.005,Z 1051.414,A -85,B 0,C 180,E1 4590.529,E2 4590.529} C_VEL
LIN {X 0,Y 107.359,Z 1050.242,A -85,B 0,C 180,E1 4586.261,E2 4586.261} C_VEL
LIN {X 0,Y 106.655,Z 1045.927,A -85,B 0,C 180,E1 4575.891,E2 4575.891} C_VEL
LIN {X 0,Y 108.209,Z 1046.066,A -85,B 0,C 180,E1 4564.892,E2 4564.892} C_VEL
LIN {X 0,Y 113.907,Z 1044.225,A -85,B 0,C 180,E1 4554.594,E2 4554.594} C_VEL
LIN {X 0,Y 123.181,Z 1040.591,A -85,B 0,C 180,E1 4545.727,E2 4545.727} C_VEL
LIN {X 0,Y 134.712,Z 1035.476,A -85,B 0,C 180,E1 4538.799,E2 4538.799} C_VEL
LIN {X 0,Y 149.046,Z 1028.275,A -85,B 0,C 180,E1 4533.011,E2 4533.011} C_VEL
LIN {X 0,Y 163.393,Z 1020.122,A -85,B 0,C 180,E1 4528.945,E2 4528.945} C_VEL
LIN {X 0,Y 168.8,Z 1016.737,A -85,B 0,C 180,E1 4527.622,E2 4527.622} C_VEL
LIN {X 0,Y 155.58,Z 1022.216,A -85,B 0,C 180,E1 4523.481,E2 4523.481} C_VEL
LIN {X 0,Y 143.519,Z 1025.57,A -85,B 0,C 180,E1 4518.649,E2 4518.649} C_VEL
LIN {X 0,Y 132.888,Z 1027.08,A -85,B 0,C 180,E1 4513.045,E2 4513.045} C_VEL
LIN {X 0,Y 123.733,Z 1026.747,A -85,B 0,C 180,E1 4506.495,E2 4506.495} C_VEL
LIN {X 0,Y 116.436,Z 1024.646,A -85,B 0,C 180,E1 4499.015,E2 4499.015} C_VEL
LIN {X 0,Y 111.236,Z 1020.599,A -85,B 0,C 180,E1 4490.688,E2 4490.688} C_VEL
LIN {X 0,Y 108.425,Z 1014.976,A -85,B 0,C 180,E1 4482.282,E2 4482.282} C_VEL
LIN {X 0,Y 107.558,Z 1007.744,A -85,B 0,C 180,E1 4474.092,E2 4474.092} C_VEL
LIN {X 0,Y 108.278,Z 998.848,A -85,B 0,C 180,E1 4466.212,E2 4466.212} C_VEL
LIN {X 0,Y 110.227,Z 988.69,A -85,B 0,C 180,E1 4459.222,E2 4459.222} C_VEL
LIN {X 0,Y 113.184,Z 976.798,A -85,B 0,C 180,E1 4452.842,E2 4452.842} C_VEL
LIN {X 0,Y 114.433,Z 972.763,A -85,B 0,C 180,E1 4450.731,E2 4450.731} C_VEL
LIN {X 0,Y 116.584,Z 972.498,A -85,B 0,C 180,E1 4448.697,E2 4448.697} C_VEL
LIN {X 0,Y 120.139,Z 971.561,A -85,B 0,C 180,E1 4446.816,E2 4446.816} C_VEL
LIN {X 0,Y 123.933,Z 971.058,A -85,B 0,C 180,E1 4444.621,E2 4444.621} C_VEL
LIN {X 0,Y 126.916,Z 970.236,A -85,B 0,C 180,E1 4443.374,E2 4443.374} C_VEL
LIN {X 0,Y 132.031,Z 969.242,A -85,B 0,C 180,E1 4441.156,E2 4441.156} C_VEL
LIN {X 0,Y 135.204,Z 968.347,A -85,B 0,C 180,E1 4440.088,E2 4440.088} C_VEL
LIN {X 0,Y 139.472,Z 967.506,A -85,B 0,C 180,E1 4438.545,E2 4438.545} C_VEL
LIN {X 0,Y 131.77,Z 980.033,A -85,B 0,C 180,E1 4433.714,E2 4433.714} C_VEL
LIN {X 0,Y 124.764,Z 990.471,A -85,B 0,C 180,E1 4428.214,E2 4428.214} C_VEL
LIN {X 0,Y 118.421,Z 999.575,A -85,B 0,C 180,E1 4421.64,E2 4421.64} C_VEL
LIN {X 0,Y 113.252,Z 1007.259,A -85,B 0,C 180,E1 4413.929,E2 4413.929} C_VEL
LIN {X 0,Y 109.82,Z 1013.322,A -85,B 0,C 180,E1 4405.301,E2 4405.301} C_VEL
LIN {X 0,Y 108.417,Z 1017.634,A -85,B 0,C 180,E1 4396.128,E2 4396.128} C_VEL
LIN {X 0,Y 109.188,Z 1020.211,A -85,B 0,C 180,E1 4386.813,E2 4386.813} C_VEL
LIN {X 0,Y 112.502,Z 1021.128,A -85,B 0,C 180,E1 4377.172,E2 4377.172} C_VEL
LIN {X 0,Y 118.015,Z 1020.245,A -85,B 0,C 180,E1 4368.638,E2 4368.638} C_VEL
LIN {X 0,Y 125.696,Z 1017.536,A -85,B 0,C 180,E1 4360.916,E2 4360.916} C_VEL
LIN {X 0,Y 135.081,Z 1012.981,A -85,B 0,C 180,E1 4354.233,E2 4354.233} C_VEL
LIN {X 0,Y 145.711,Z 1006.601,A -85,B 0,C 180,E1 4348.561,E2 4348.561} C_VEL
LIN {X 0,Y 156.532,Z 998.811,A -85,B 0,C 180,E1 4344.02,E2 4344.02} C_VEL
LIN {X 0,Y 167.475,Z 989.459,A -85,B 0,C 180,E1 4340.26,E2 4340.26} C_VEL
LIN {X 0,Y 178.362,Z 978.411,A -85,B 0,C 180,E1 4337.103,E2 4337.103} C_VEL
LIN {X 0,Y 188.955,Z 965.682,A -85,B 0,C 180,E1 4334.457,E2 4334.457} C_VEL
LIN {X 0,Y 198.549,Z 951.876,A -85,B 0,C 180,E1 4332.328,E2 4332.328} C_VEL
LIN {X 0,Y 207.055,Z 936.962,A -85,B 0,C 180,E1 4330.604,E2 4330.604} C_VEL
LIN {X 0,Y 214.241,Z 921.16,A -85,B 0,C 180,E1 4329.228,E2 4329.228} C_VEL
LIN {X 0,Y 220.172,Z 904.231,A -85,B 0,C 180,E1 4328.116,E2 4328.116} C_VEL
LIN {X 0,Y 224.554,Z 886.777,A -85,B 0,C 180,E1 4327.272,E2 4327.272} C_VEL
LIN {X 0,Y 227.346,Z 868.842,A -85,B 0,C 180,E1 4326.665,E2 4326.665} C_VEL
LIN {X 0,Y 233.144,Z 816.992,A -85,B 0,C 180,E1 4325.489,E2 4325.489} C_VEL
LIN {X 0,Y 231.863,Z 813.283,A -85,B 0,C 180,E1 4322.843,E2 4322.843} C_VEL
LIN {X 0,Y 230.871,Z 810.368,A -85,B 0,C 180,E1 4319.752,E2 4319.752} C_VEL
LIN {X 0,Y 230.412,Z 808.769,A -85,B 0,C 180,E1 4315.77,E2 4315.77} C_VEL
LIN {X 0,Y 230.581,Z 809.308,A -85,B 0,C 180,E1 4312.776,E2 4312.776} C_VEL
LIN {X 0,Y 231.53,Z 811.846,A -85,B 0,C 180,E1 4309.047,E2 4309.047} C_VEL
LIN {X 0,Y 233.076,Z 816.003,A -85,B 0,C 180,E1 4305.657,E2 4305.657} C_VEL
LIN {X 0,Y 233.348,Z 817.269,A -85,B 0,C 180,E1 4305.086,E2 4305.086} C_VEL
LIN {X 0,Y 225.203,Z 887.66,A -85,B 0,C 180,E1 4303.619,E2 4303.619} C_VEL
LIN {X 0,Y 221.286,Z 906.073,A -85,B 0,C 180,E1 4303.092,E2 4303.092} C_VEL
LIN {X 0,Y 215.564,Z 924.333,A -85,B 0,C 180,E1 4302.396,E2 4302.396} C_VEL
LIN {X 0,Y 208.707,Z 940.837,A -85,B 0,C 180,E1 4301.542,E2 4301.542} C_VEL
LIN {X 0,Y 203.118,Z 951.974,A -85,B 0,C 180,E1 4300.786,E2 4300.786} C_VEL
LIN {X 0,Y 199.061,Z 958.638,A -85,B 0,C 180,E1 4300.515,E2 4300.515} C_VEL
LIN {X 0,Y 188.126,Z 972.752,A -85,B 0,C 180,E1 4300.623,E2 4300.623} C_VEL
LIN {X 0,Y 183.252,Z 978.669,A -85,B 0,C 180,E1 4300.32,E2 4300.32} C_VEL
LIN {X 0,Y 181.932,Z 980.299,A -85,B 0,C 180,E1 4300.126,E2 4300.126} C_VEL
LIN {X 0,Y 170.475,Z 993.852,A -85,B 0,C 180,E1 4297.923,E2 4297.923} C_VEL
LIN {X 0,Y 158.665,Z 1005.912,A -85,B 0,C 180,E1 4295.153,E2 4295.153} C_VEL
LIN {X 0,Y 146.599,Z 1016.655,A -85,B 0,C 180,E1 4291.62,E2 4291.62} C_VEL
LIN {X 0,Y 133.857,Z 1026.638,A -85,B 0,C 180,E1 4286.78,E2 4286.78} C_VEL
LIN {X 0,Y 121.792,Z 1035.001,A -85,B 0,C 180,E1 4280.505,E2 4280.505} C_VEL
LIN {X 0,Y 111.348,Z 1041.622,A -85,B 0,C 180,E1 4272.582,E2 4272.582} C_VEL
LIN {X 0,Y 103.174,Z 1046.628,A -85,B 0,C 180,E1 4262.531,E2 4262.531} C_VEL
LIN {X 0,Y 98.788,Z 1049.622,A -85,B 0,C 180,E1 4251.367,E2 4251.367} C_VEL
LIN {X 0,Y 98.188,Z 1050.71,A -85,B 0,C 180,E1 4239.967,E2 4239.967} C_VEL
LIN {X 0,Y 100.054,Z 1050.096,A -85,B 0,C 180,E1 4230.571,E2 4230.571} C_VEL
LIN {X 0,Y 99.244,Z 1048.685,A -85,B 0,C 180,E1 4225.376,E2 4225.376} C_VEL
LIN {X 0,Y 98.768,Z 1044.552,A -85,B 0,C 180,E1 4215.338,E2 4215.338} C_VEL
LIN {X 0,Y 98.922,Z 1044.045,A -85,B 0,C 180,E1 4213.558,E2 4213.558} C_VEL
LIN {X 0,Y 101.385,Z 1044.323,A -85,B 0,C 180,E1 4201.744,E2 4201.744} C_VEL
LIN {X 0,Y 108.214,Z 1042.757,A -85,B 0,C 180,E1 4191.074,E2 4191.074} C_VEL
LIN {X 0,Y 118.655,Z 1039.366,A -85,B 0,C 180,E1 4182.135,E2 4182.135} C_VEL
LIN {X 0,Y 131.909,Z 1034.312,A -85,B 0,C 180,E1 4175.05,E2 4175.05} C_VEL
LIN {X 0,Y 146.423,Z 1027.885,A -85,B 0,C 180,E1 4169.86,E2 4169.86} C_VEL
LIN {X 0,Y 155.882,Z 1023.122,A -85,B 0,C 180,E1 4167.291,E2 4167.291} C_VEL
LIN {X 0,Y 142.504,Z 1026.86,A -85,B 0,C 180,E1 4162.699,E2 4162.699} C_VEL
LIN {X 0,Y 129.987,Z 1028.617,A -85,B 0,C 180,E1 4156.995,E2 4156.995} C_VEL
LIN {X 0,Y 119.725,Z 1028.434,A -85,B 0,C 180,E1 4150.586,E2 4150.586} C_VEL
LIN {X 0,Y 110.809,Z 1026.276,A -85,B 0,C 180,E1 4142.585,E2 4142.585} C_VEL
LIN {X 0,Y 104.584,Z 1022.262,A -85,B 0,C 180,E1 4133.879,E2 4133.879} C_VEL
LIN {X 0,Y 100.874,Z 1016.364,A -85,B 0,C 180,E1 4124.476,E2 4124.476} C_VEL
LIN {X 0,Y 99.593,Z 1009.152,A -85,B 0,C 180,E1 4115.692,E2 4115.692} C_VEL
LIN {X 0,Y 100.098,Z 1000.163,A -85,B 0,C 180,E1 4107.044,E2 4107.044} C_VEL
LIN {X 0,Y 102.204,Z 989.087,A -85,B 0,C 180,E1 4098.879,E2 4098.879} C_VEL
LIN {X 0,Y 104.815,Z 979.221,A -85,B 0,C 180,E1 4092.932,E2 4092.932} C_VEL
LIN {X 0,Y 106.181,Z 978.977,A -85,B 0,C 180,E1 4091.119,E2 4091.119} C_VEL
LIN {X 0,Y 109.97,Z 978.124,A -85,B 0,C 180,E1 4088.562,E2 4088.562} C_VEL
LIN {X 0,Y 113.652,Z 977.745,A -85,B 0,C 180,E1 4085.963,E2 4085.963} C_VEL
LIN {X 0,Y 116.476,Z 977.101,A -85,B 0,C 180,E1 4084.502,E2 4084.502} C_VEL
LIN {X 0,Y 121.433,Z 976.236,A -85,B 0,C 180,E1 4081.994,E2 4081.994} C_VEL
LIN {X 0,Y 124.437,Z 975.614,A -85,B 0,C 180,E1 4080.709,E2 4080.709} C_VEL
LIN {X 0,Y 129.79,Z 974.551,A -85,B 0,C 180,E1 4078.61,E2 4078.61} C_VEL
LIN {X 0,Y 121.759,Z 986.364,A -85,B 0,C 180,E1 4073.215,E2 4073.215} C_VEL
LIN {X 0,Y 114.373,Z 996.429,A -85,B 0,C 180,E1 4066.769,E2 4066.769} C_VEL
LIN {X 0,Y 108.033,Z 1004.993,A -85,B 0,C 180,E1 4059.054,E2 4059.054} C_VEL
LIN {X 0,Y 103.53,Z 1011.653,A -85,B 0,C 180,E1 4050.555,E2 4050.555} C_VEL
LIN {X 0,Y 100.916,Z 1016.893,A -85,B 0,C 180,E1 4040.88,E2 4040.88} C_VEL
LIN {X 0,Y 100.661,Z 1020.368,A -85,B 0,C 180,E1 4030.674,E2 4030.674} C_VEL
LIN {X 0,Y 103.03,Z 1022.135,A -85,B 0,C 180,E1 4020.336,E2 4020.336} C_VEL
LIN {X 0,Y 107.877,Z 1022.127,A -85,B 0,C 180,E1 4010.933,E2 4010.933} C_VEL
LIN {X 0,Y 115.114,Z 1020.381,A -85,B 0,C 180,E1 4002.416,E2 4002.416} C_VEL
LIN {X 0,Y 124.437,Z 1016.728,A -85,B 0,C 180,E1 3994.96,E2 3994.96} C_VEL
LIN {X 0,Y 135.121,Z 1011.295,A -85,B 0,C 180,E1 3988.751,E2 3988.751} C_VEL
LIN {X 0,Y 146.365,Z 1004.293,A -85,B 0,C 180,E1 3983.741,E2 3983.741} C_VEL
LIN {X 0,Y 158.106,Z 995.542,A -85,B 0,C 180,E1 3979.565,E2 3979.565} C_VEL
LIN {X 0,Y 169.684,Z 985.18,A -85,B 0,C 180,E1 3976.166,E2 3976.166} C_VEL
LIN {X 0,Y 180.526,Z 973.656,A -85,B 0,C 180,E1 3973.452,E2 3973.452} C_VEL
LIN {X 0,Y 190.914,Z 960.494,A -85,B 0,C 180,E1 3971.174,E2 3971.174} C_VEL
LIN {X 0,Y 200.131,Z 946.422,A -85,B 0,C 180,E1 3969.354,E2 3969.354} C_VEL
LIN {X 0,Y 207.954,Z 931.828,A -85,B 0,C 180,E1 3967.923,E2 3967.923} C_VEL
LIN {X 0,Y 214.75,Z 915.846,A -85,B 0,C 180,E1 3966.727,E2 3966.727} C_VEL
LIN {X 0,Y 220.211,Z 898.754,A -85,B 0,C 180,E1 3965.765,E2 3965.765} C_VEL
LIN {X 0,Y 224.201,Z 880.525,A -85,B 0,C 180,E1 3965.02,E2 3965.02} C_VEL
LIN {X 0,Y 227.609,Z 853.35,A -85,B 0,C 180,E1 3964.308,E2 3964.308} C_VEL
LIN {X 0,Y 231.152,Z 822.604,A -85,B 0,C 180,E1 3963.659,E2 3963.659} C_VEL
LIN {X 0,Y 230.334,Z 820.231,A -85,B 0,C 180,E1 3961.617,E2 3961.617} C_VEL
LIN {X 0,Y 229.744,Z 818.112,A -85,B 0,C 180,E1 3959.252,E2 3959.252} C_VEL
LIN {X 0,Y 229.407,Z 816.705,A -85,B 0,C 180,E1 3955.751,E2 3955.751} C_VEL
LIN {X 0,Y 229.542,Z 817.194,A -85,B 0,C 180,E1 3952.995,E2 3952.995} C_VEL
LIN {X 0,Y 230.338,Z 819.556,A -85,B 0,C 180,E1 3949.496,E2 3949.496} C_VEL
LIN {X 0,Y 231.357,Z 822.596,A -85,B 0,C 180,E1 3946.928,E2 3946.928} C_VEL
LIN {X 0,Y 223.707,Z 886.892,A -85,B 0,C 180,E1 3945.64,E2 3945.64} C_VEL
LIN {X 0,Y 219.686,Z 905.394,A -85,B 0,C 180,E1 3945.144,E2 3945.144} C_VEL
LIN {X 0,Y 214.221,Z 922.636,A -85,B 0,C 180,E1 3944.539,E2 3944.539} C_VEL
